DATA_BLOCK "DB00800_St_ConstAiRawData"   // DB800
TITLE = Static DB [SYSTEM CONSTANTS] — Analog Input Card Types, Ranges and Coefficients
{ S7_Optimized_Access := 'TRUE' }
AUTHOR : M_Gledhill
FAMILY : SysConstants
NAME : St_ConstAiRawData
VERSION : 1.0
// PRACTICAL SERIES AUTOMATION LIBRARY (PAL)   —   COPYRIGHT 2020 – M. GLEDHILL (MIT LICENCE)
//                   ———— ◆ ————
// FULL ONLINE DOCUMENTATION IS AVAILABLE AT: https://practicalseries.com/2001-pal/index.html
// stored: AutoNumber false, DBAccessibleFromOPCUA true, IsOnlyStoredInLoadMemory false, IsRetainMemResEnabled false, IsWriteProtectedInAS true, MemoryReserve 100
   VAR
      _DB_Header { ExternalAccessible := 'False'; ExternalVisible := 'False'; ExternalWritable := 'False'} : Array[0..79] of Bool;   // Static DB [SYSTEM CONSTANTS] — Analog Input Card Types, Ranges and Coefficients
      __________0000_0 { ExternalAccessible := 'False'; ExternalVisible := 'False'; ExternalWritable := 'False'} : Bool := false;
      __________0000_1 { ExternalAccessible := 'False'; ExternalVisible := 'False'; ExternalWritable := 'False'} : Bool := false;
      revInfo { ExternalWritable := 'False'} : "UT01000_St_SysRevision";
      __________0010_0 { ExternalAccessible := 'False'; ExternalVisible := 'False'; ExternalWritable := 'False'} : Bool := false;
      __________0010_1 { ExternalAccessible := 'False'; ExternalVisible := 'False'; ExternalWritable := 'False'} : Bool := false;
      AI_0000 { ExternalWritable := 'False'} : "UT00800_St_ConstAiRawData";
      __________0020_0 { ExternalAccessible := 'False'; ExternalVisible := 'False'; ExternalWritable := 'False'} : Bool := false;
      __________0020_1 { ExternalAccessible := 'False'; ExternalVisible := 'False'; ExternalWritable := 'False'} : Bool := false;   // ▀▀▀▀ ANALOG INPUT SIGNAL — VOLTAGE
      AI_1000 { ExternalWritable := 'False'} : "UT00800_St_ConstAiRawData";   // AI Voltage (-25 mV to +25 mV)
      AI_1001 { ExternalWritable := 'False'} : "UT00800_St_ConstAiRawData";   // AI Voltage (-50 mV to +50 mV)
      AI_1002 { ExternalWritable := 'False'} : "UT00800_St_ConstAiRawData";   // AI Voltage (-80 mV to +80 mV)
      AI_1003 { ExternalWritable := 'False'} : "UT00800_St_ConstAiRawData";   // AI Voltage (-250 mV to +250 mV)
      AI_1004 { ExternalWritable := 'False'} : "UT00800_St_ConstAiRawData";   // AI Voltage (-500 mV to +500 mV)
      AI_1005 { ExternalWritable := 'False'} : "UT00800_St_ConstAiRawData";   // AI Voltage (-1 V to +1 V)
      AI_1007 { ExternalWritable := 'False'} : "UT00800_St_ConstAiRawData";   // AI Voltage (-2.5 V to +2.5 V)
      AI_1008 { ExternalWritable := 'False'} : "UT00800_St_ConstAiRawData";   // AI Voltage (-5 V to +5 V)
      AI_1009 { ExternalWritable := 'False'} : "UT00800_St_ConstAiRawData";   // AI Voltage (-10 V to +10 V)
      AI_100A { ExternalWritable := 'False'} : "UT00800_St_ConstAiRawData";   // AI Voltage (1 V to 5 V)
      __________0030_0 { ExternalAccessible := 'False'; ExternalVisible := 'False'; ExternalWritable := 'False'} : Bool := false;
      __________0030_1 { ExternalAccessible := 'False'; ExternalVisible := 'False'; ExternalWritable := 'False'} : Bool := false;   // ▀▀▀▀ ANALOG INPUT SIGNAL — CURRENT (4 WIRE)
      AI_2002 { ExternalWritable := 'False'} : "UT00800_St_ConstAiRawData";   // AI Current - 4-wire (0 mA to 20 mA)
      AI_2003 { ExternalWritable := 'False'} : "UT00800_St_ConstAiRawData";   // AI Current - 4-wire (4 mA to 20 mA)
      AI_2004 { ExternalWritable := 'False'} : "UT00800_St_ConstAiRawData";   // AI Current - 4-wire (-20 mA to +20 mA)
      __________0040_0 { ExternalAccessible := 'False'; ExternalVisible := 'False'; ExternalWritable := 'False'} : Bool := false;
      __________0040_1 { ExternalAccessible := 'False'; ExternalVisible := 'False'; ExternalWritable := 'False'} : Bool := false;   // ▀▀▀▀ ANALOG INPUT SIGNAL — CURRENT (2 WIRE)
      AI_3003 { ExternalWritable := 'False'} : "UT00800_St_ConstAiRawData";   // AI Current - 2-wire (4 mA to 20 mA)
      __________0050_0 { ExternalAccessible := 'False'; ExternalVisible := 'False'; ExternalWritable := 'False'} : Bool := false;
      __________0050_1 { ExternalAccessible := 'False'; ExternalVisible := 'False'; ExternalWritable := 'False'} : Bool := false;   // ▀▀▀▀ ANALOG INPUT SIGNAL — RESISTANCE (4 WIRE)
      AI_4001 { ExternalWritable := 'False'} : "UT00800_St_ConstAiRawData";   // AI Resistance - 4-wire (150 Ohm)
      AI_4002 { ExternalWritable := 'False'} : "UT00800_St_ConstAiRawData";   // AI Resistance - 4-wire (300 Ohm)
      AI_4003 { ExternalWritable := 'False'} : "UT00800_St_ConstAiRawData";   // AI Resistance - 4-wire (600 Ohm)
      AI_4005 { ExternalWritable := 'False'} : "UT00800_St_ConstAiRawData";   // AI Resistance - 4-wire (6000 Ohm)
      __________0060_0 { ExternalAccessible := 'False'; ExternalVisible := 'False'; ExternalWritable := 'False'} : Bool := false;
      __________0060_1 { ExternalAccessible := 'False'; ExternalVisible := 'False'; ExternalWritable := 'False'} : Bool := false;   // ▀▀▀▀ ANALOG INPUT SIGNAL — RESISTANCE (3 WIRE)
      AI_5001 { ExternalWritable := 'False'} : "UT00800_St_ConstAiRawData";   // AI Resistance - 3-wire (150 Ohm)
      AI_5002 { ExternalWritable := 'False'} : "UT00800_St_ConstAiRawData";   // AI Resistance - 3-wire (300 Ohm)
      AI_5003 { ExternalWritable := 'False'} : "UT00800_St_ConstAiRawData";   // AI Resistance - 3-wire (600 Ohm)
      AI_5005 { ExternalWritable := 'False'} : "UT00800_St_ConstAiRawData";   // AI Resistance - 3-wire (6000 Ohm)
      __________0070_0 { ExternalAccessible := 'False'; ExternalVisible := 'False'; ExternalWritable := 'False'} : Bool := false;
      __________0070_1 { ExternalAccessible := 'False'; ExternalVisible := 'False'; ExternalWritable := 'False'} : Bool := false;   // ▀▀▀▀ ANALOG INPUT SIGNAL — RESISTANCE (2 WIRE)
      AI_6001 { ExternalWritable := 'False'} : "UT00800_St_ConstAiRawData";   // AI Resistance - 2-wire (150 Ohm)
      AI_6002 { ExternalWritable := 'False'} : "UT00800_St_ConstAiRawData";   // AI Resistance - 2-wire (300 Ohm)
      AI_6003 { ExternalWritable := 'False'} : "UT00800_St_ConstAiRawData";   // AI Resistance - 2-wire (600 Ohm)
      AI_6005 { ExternalWritable := 'False'} : "UT00800_St_ConstAiRawData";   // AI Resistance - 2-wire (6000 Ohm)
      AI_600F { ExternalWritable := 'False'} : "UT00800_St_ConstAiRawData";   // AI Resistance - 2-wire (PTC)
      __________0080_0 { ExternalAccessible := 'False'; ExternalVisible := 'False'; ExternalWritable := 'False'} : Bool := false;
      __________0080_1 { ExternalAccessible := 'False'; ExternalVisible := 'False'; ExternalWritable := 'False'} : Bool := false;   // ▀▀▀▀ ANALOG INPUT SIGNAL — THERMAL RESISTANCE (4 WIRE) Cu x0
      AI_7B0E { ExternalWritable := 'False'} : "UT00800_St_ConstAiRawData";   // AI Thermal Resistance - 4-wire (Cu10 climate - 426)
      AI_7C0E { ExternalWritable := 'False'} : "UT00800_St_ConstAiRawData";   // AI Thermal Resistance - 4-wire (Cu10 climate - 427)
      AI_7D0E { ExternalWritable := 'False'} : "UT00800_St_ConstAiRawData";   // AI Thermal Resistance - 4-wire (Cu10 climate - 428)
      AI_7B0F { ExternalWritable := 'False'} : "UT00800_St_ConstAiRawData";   // AI Thermal Resistance - 4-wire (Cu10 standard - 426)
      AI_7C0F { ExternalWritable := 'False'} : "UT00800_St_ConstAiRawData";   // AI Thermal Resistance - 4-wire (Cu10 standard - 427)
      AI_7D0F { ExternalWritable := 'False'} : "UT00800_St_ConstAiRawData";   // AI Thermal Resistance - 4-wire (Cu10 standard - 428)
      AI_7B19 { ExternalWritable := 'False'} : "UT00800_St_ConstAiRawData";   // AI Thermal Resistance - 4-wire (Cu50 climate - 426)
      AI_7C19 { ExternalWritable := 'False'} : "UT00800_St_ConstAiRawData";   // AI Thermal Resistance - 4-wire (Cu50 climate - 427)
      AI_7D19 { ExternalWritable := 'False'} : "UT00800_St_ConstAiRawData";   // AI Thermal Resistance - 4-wire (Cu50 climate - 428)
      AI_7B18 { ExternalWritable := 'False'} : "UT00800_St_ConstAiRawData";   // AI Thermal Resistance - 4-wire (Cu50 standard - 426)
      AI_7C18 { ExternalWritable := 'False'} : "UT00800_St_ConstAiRawData";   // AI Thermal Resistance - 4-wire (Cu50 standard - 427)
      AI_7D18 { ExternalWritable := 'False'} : "UT00800_St_ConstAiRawData";   // AI Thermal Resistance - 4-wire (Cu50 standard - 428)
      AI_7B1B { ExternalWritable := 'False'} : "UT00800_St_ConstAiRawData";   // AI Thermal Resistance - 4-wire (Cu100 climate - 426)
      AI_7C1B { ExternalWritable := 'False'} : "UT00800_St_ConstAiRawData";   // AI Thermal Resistance - 4-wire (Cu100 climate - 427)
      AI_7D1B { ExternalWritable := 'False'} : "UT00800_St_ConstAiRawData";   // AI Thermal Resistance - 4-wire (Cu100 climate - 428)
      AI_7B1A { ExternalWritable := 'False'} : "UT00800_St_ConstAiRawData";   // AI Thermal Resistance - 4-wire (Cu100 standard - 426)
      AI_7C1A { ExternalWritable := 'False'} : "UT00800_St_ConstAiRawData";   // AI Thermal Resistance - 4-wire (Cu100 standard - 427)
      AI_7D1A { ExternalWritable := 'False'} : "UT00800_St_ConstAiRawData";   // AI Thermal Resistance - 4-wire (Cu100 standard - 428)
      __________0090_0 { ExternalAccessible := 'False'; ExternalVisible := 'False'; ExternalWritable := 'False'} : Bool := false;
      __________0090_1 { ExternalAccessible := 'False'; ExternalVisible := 'False'; ExternalWritable := 'False'} : Bool := false;   // ▀▀▀▀ ANALOG INPUT SIGNAL — THERMAL RESISTANCE (4 WIRE) LG-Ni x0
      AI_7A1D { ExternalWritable := 'False'} : "UT00800_St_ConstAiRawData";   // AI Thermal Resistance - 4-wire (LG-Ni1000 climate - 500)
      AI_7A1C { ExternalWritable := 'False'} : "UT00800_St_ConstAiRawData";   // AI Thermal Resistance - 4-wire (LG-Ni1000 standard - 500)
      __________0100_0 { ExternalAccessible := 'False'; ExternalVisible := 'False'; ExternalWritable := 'False'} : Bool := false;
      __________0100_1 { ExternalAccessible := 'False'; ExternalVisible := 'False'; ExternalWritable := 'False'} : Bool := false;   // ▀▀▀▀ ANALOG INPUT SIGNAL — THERMAL RESISTANCE (4 WIRE) Ni x0
      AI_771F { ExternalWritable := 'False'} : "UT00800_St_ConstAiRawData";   // AI Thermal Resistance - 4-wire (Ni10 climate - 617)
      AI_781F { ExternalWritable := 'False'} : "UT00800_St_ConstAiRawData";   // AI Thermal Resistance - 4-wire (Ni10 climate - 618)
      AI_791F { ExternalWritable := 'False'} : "UT00800_St_ConstAiRawData";   // AI Thermal Resistance - 4-wire (Ni10 climate - 672)
      AI_771E { ExternalWritable := 'False'} : "UT00800_St_ConstAiRawData";   // AI Thermal Resistance - 4-wire (Ni10 standard - 617)
      AI_781E { ExternalWritable := 'False'} : "UT00800_St_ConstAiRawData";   // AI Thermal Resistance - 4-wire (Ni10 standard - 618)
      AI_791E { ExternalWritable := 'False'} : "UT00800_St_ConstAiRawData";   // AI Thermal Resistance - 4-wire (Ni10 standard - 672)
      AI_770D { ExternalWritable := 'False'} : "UT00800_St_ConstAiRawData";   // AI Thermal Resistance - 4-wire (Ni120 climate - 617)
      AI_780D { ExternalWritable := 'False'} : "UT00800_St_ConstAiRawData";   // AI Thermal Resistance - 4-wire (Ni120 climate - 618)
      AI_790D { ExternalWritable := 'False'} : "UT00800_St_ConstAiRawData";   // AI Thermal Resistance - 4-wire (Ni120 climate - 672)
      AI_770C { ExternalWritable := 'False'} : "UT00800_St_ConstAiRawData";   // AI Thermal Resistance - 4-wire (Ni120 standard - 617)
      AI_780C { ExternalWritable := 'False'} : "UT00800_St_ConstAiRawData";   // AI Thermal Resistance - 4-wire (Ni120 standard - 618)
      AI_790C { ExternalWritable := 'False'} : "UT00800_St_ConstAiRawData";   // AI Thermal Resistance - 4-wire (Ni120 standard - 672)
      AI_7701 { ExternalWritable := 'False'} : "UT00800_St_ConstAiRawData";   // AI Thermal Resistance - 4-wire (Ni100 climate - 617)
      AI_7801 { ExternalWritable := 'False'} : "UT00800_St_ConstAiRawData";   // AI Thermal Resistance - 4-wire (Ni100 climate - 618)
      AI_7901 { ExternalWritable := 'False'} : "UT00800_St_ConstAiRawData";   // AI Thermal Resistance - 4-wire (Ni100 climate - 672)
      AI_7703 { ExternalWritable := 'False'} : "UT00800_St_ConstAiRawData";   // AI Thermal Resistance - 4-wire (Ni100 standard - 617)
      AI_7803 { ExternalWritable := 'False'} : "UT00800_St_ConstAiRawData";   // AI Thermal Resistance - 4-wire (Ni100 standard - 618)
      AI_7903 { ExternalWritable := 'False'} : "UT00800_St_ConstAiRawData";   // AI Thermal Resistance - 4-wire (Ni100 standard - 672)
      AI_7711 { ExternalWritable := 'False'} : "UT00800_St_ConstAiRawData";   // AI Thermal Resistance - 4-wire (Ni200 climate - 617)
      AI_7811 { ExternalWritable := 'False'} : "UT00800_St_ConstAiRawData";   // AI Thermal Resistance - 4-wire (Ni200 climate - 618)
      AI_7911 { ExternalWritable := 'False'} : "UT00800_St_ConstAiRawData";   // AI Thermal Resistance - 4-wire (Ni200 climate - 672)
      AI_7710 { ExternalWritable := 'False'} : "UT00800_St_ConstAiRawData";   // AI Thermal Resistance - 4-wire (Ni200 standard - 617)
      AI_7810 { ExternalWritable := 'False'} : "UT00800_St_ConstAiRawData";   // AI Thermal Resistance - 4-wire (Ni200 standard - 618)
      AI_7910 { ExternalWritable := 'False'} : "UT00800_St_ConstAiRawData";   // AI Thermal Resistance - 4-wire (Ni200 standard - 672)
      AI_7713 { ExternalWritable := 'False'} : "UT00800_St_ConstAiRawData";   // AI Thermal Resistance - 4-wire (Ni500 climate - 617)
      AI_7813 { ExternalWritable := 'False'} : "UT00800_St_ConstAiRawData";   // AI Thermal Resistance - 4-wire (Ni500 climate - 618)
      AI_7913 { ExternalWritable := 'False'} : "UT00800_St_ConstAiRawData";   // AI Thermal Resistance - 4-wire (Ni500 climate - 672)
      AI_7712 { ExternalWritable := 'False'} : "UT00800_St_ConstAiRawData";   // AI Thermal Resistance - 4-wire (Ni500 standard - 617)
      AI_7812 { ExternalWritable := 'False'} : "UT00800_St_ConstAiRawData";   // AI Thermal Resistance - 4-wire (Ni500 standard - 618)
      AI_7912 { ExternalWritable := 'False'} : "UT00800_St_ConstAiRawData";   // AI Thermal Resistance - 4-wire (Ni500 standard - 672)
      AI_770A { ExternalWritable := 'False'} : "UT00800_St_ConstAiRawData";   // AI Thermal Resistance - 4-wire (Ni1000 climate - 617)
      AI_780A { ExternalWritable := 'False'} : "UT00800_St_ConstAiRawData";   // AI Thermal Resistance - 4-wire (Ni1000 climate - 618)
      AI_790A { ExternalWritable := 'False'} : "UT00800_St_ConstAiRawData";   // AI Thermal Resistance - 4-wire (Ni1000 climate - 672)
      AI_7706 { ExternalWritable := 'False'} : "UT00800_St_ConstAiRawData";   // AI Thermal Resistance - 4-wire (Ni1000 standard - 617)
      AI_7806 { ExternalWritable := 'False'} : "UT00800_St_ConstAiRawData";   // AI Thermal Resistance - 4-wire (Ni1000 standard - 618)
      AI_7906 { ExternalWritable := 'False'} : "UT00800_St_ConstAiRawData";   // AI Thermal Resistance - 4-wire (Ni1000 standard - 672)
      __________0110_0 { ExternalAccessible := 'False'; ExternalVisible := 'False'; ExternalWritable := 'False'} : Bool := false;
      __________0110_1 { ExternalAccessible := 'False'; ExternalVisible := 'False'; ExternalWritable := 'False'} : Bool := false;   // ▀▀▀▀ ANALOG INPUT SIGNAL — THERMAL RESISTANCE (4 WIRE) Pt x0
      AI_7015 { ExternalWritable := 'False'} : "UT00800_St_ConstAiRawData";   // AI Thermal Resistance - 4-wire (Pt10 climate - 3851)
      AI_7215 { ExternalWritable := 'False'} : "UT00800_St_ConstAiRawData";   // AI Thermal Resistance - 4-wire (Pt10 climate - 3902)
      AI_7515 { ExternalWritable := 'False'} : "UT00800_St_ConstAiRawData";   // AI Thermal Resistance - 4-wire (Pt10 climate - 391)
      AI_7115 { ExternalWritable := 'False'} : "UT00800_St_ConstAiRawData";   // AI Thermal Resistance - 4-wire (Pt10 climate - 3916)
      AI_7315 { ExternalWritable := 'False'} : "UT00800_St_ConstAiRawData";   // AI Thermal Resistance - 4-wire (Pt10 climate - 392)
      AI_7014 { ExternalWritable := 'False'} : "UT00800_St_ConstAiRawData";   // AI Thermal Resistance - 4-wire (Pt10 standard - 3851)
      AI_7214 { ExternalWritable := 'False'} : "UT00800_St_ConstAiRawData";   // AI Thermal Resistance - 4-wire (Pt10 standard - 3902)
      AI_7514 { ExternalWritable := 'False'} : "UT00800_St_ConstAiRawData";   // AI Thermal Resistance - 4-wire (Pt10 standard - 391)
      AI_7114 { ExternalWritable := 'False'} : "UT00800_St_ConstAiRawData";   // AI Thermal Resistance - 4-wire (Pt10 standard - 3916)
      AI_7314 { ExternalWritable := 'False'} : "UT00800_St_ConstAiRawData";   // AI Thermal Resistance - 4-wire (Pt10 standard - 392)
      AI_7017 { ExternalWritable := 'False'} : "UT00800_St_ConstAiRawData";   // AI Thermal Resistance - 4-wire (Pt50 climate - 3851)
      AI_7217 { ExternalWritable := 'False'} : "UT00800_St_ConstAiRawData";   // AI Thermal Resistance - 4-wire (Pt50 climate - 3902)
      AI_7517 { ExternalWritable := 'False'} : "UT00800_St_ConstAiRawData";   // AI Thermal Resistance - 4-wire (Pt50 climate - 391)
      AI_7117 { ExternalWritable := 'False'} : "UT00800_St_ConstAiRawData";   // AI Thermal Resistance - 4-wire (Pt50 climate - 3916)
      AI_7317 { ExternalWritable := 'False'} : "UT00800_St_ConstAiRawData";   // AI Thermal Resistance - 4-wire (Pt50 climate - 392)
      AI_7016 { ExternalWritable := 'False'} : "UT00800_St_ConstAiRawData";   // AI Thermal Resistance - 4-wire (Pt50 standard - 3851)
      AI_7216 { ExternalWritable := 'False'} : "UT00800_St_ConstAiRawData";   // AI Thermal Resistance - 4-wire (Pt50 standard - 3902)
      AI_7516 { ExternalWritable := 'False'} : "UT00800_St_ConstAiRawData";   // AI Thermal Resistance - 4-wire (Pt50 standard - 391)
      AI_7116 { ExternalWritable := 'False'} : "UT00800_St_ConstAiRawData";   // AI Thermal Resistance - 4-wire (Pt50 standard - 3916)
      AI_7316 { ExternalWritable := 'False'} : "UT00800_St_ConstAiRawData";   // AI Thermal Resistance - 4-wire (Pt50 standard - 392)
      AI_7000 { ExternalWritable := 'False'} : "UT00800_St_ConstAiRawData";   // AI Thermal Resistance - 4-wire (Pt100 climate - 3851)
      AI_7200 { ExternalWritable := 'False'} : "UT00800_St_ConstAiRawData";   // AI Thermal Resistance - 4-wire (Pt100 climate - 3902)
      AI_7500 { ExternalWritable := 'False'} : "UT00800_St_ConstAiRawData";   // AI Thermal Resistance - 4-wire (Pt100 climate - 391)
      AI_7100 { ExternalWritable := 'False'} : "UT00800_St_ConstAiRawData";   // AI Thermal Resistance - 4-wire (Pt100 climate - 3916)
      AI_7300 { ExternalWritable := 'False'} : "UT00800_St_ConstAiRawData";   // AI Thermal Resistance - 4-wire (Pt100 climate - 392)
      AI_7002 { ExternalWritable := 'False'} : "UT00800_St_ConstAiRawData";   // AI Thermal Resistance - 4-wire (Pt100 standard - 3851)
      AI_7202 { ExternalWritable := 'False'} : "UT00800_St_ConstAiRawData";   // AI Thermal Resistance - 4-wire (Pt100 standard - 3902)
      AI_7502 { ExternalWritable := 'False'} : "UT00800_St_ConstAiRawData";   // AI Thermal Resistance - 4-wire (Pt100 standard - 391)
      AI_7102 { ExternalWritable := 'False'} : "UT00800_St_ConstAiRawData";   // AI Thermal Resistance - 4-wire (Pt100 standard - 3916)
      AI_7302 { ExternalWritable := 'False'} : "UT00800_St_ConstAiRawData";   // AI Thermal Resistance - 4-wire (Pt100 standard - 392)
      AI_7007 { ExternalWritable := 'False'} : "UT00800_St_ConstAiRawData";   // AI Thermal Resistance - 4-wire (Pt200 climate - 3851)
      AI_7207 { ExternalWritable := 'False'} : "UT00800_St_ConstAiRawData";   // AI Thermal Resistance - 4-wire (Pt200 climate - 3902)
      AI_7507 { ExternalWritable := 'False'} : "UT00800_St_ConstAiRawData";   // AI Thermal Resistance - 4-wire (Pt200 climate - 391)
      AI_7107 { ExternalWritable := 'False'} : "UT00800_St_ConstAiRawData";   // AI Thermal Resistance - 4-wire (Pt200 climate - 3916)
      AI_7307 { ExternalWritable := 'False'} : "UT00800_St_ConstAiRawData";   // AI Thermal Resistance - 4-wire (Pt200 climate - 392)
      AI_700B { ExternalWritable := 'False'} : "UT00800_St_ConstAiRawData";   // AI Thermal Resistance - 4-wire (Pt200 standard - 3851)
      AI_720B { ExternalWritable := 'False'} : "UT00800_St_ConstAiRawData";   // AI Thermal Resistance - 4-wire (Pt200 standard - 3902)
      AI_750B { ExternalWritable := 'False'} : "UT00800_St_ConstAiRawData";   // AI Thermal Resistance - 4-wire (Pt200 standard - 391)
      AI_710B { ExternalWritable := 'False'} : "UT00800_St_ConstAiRawData";   // AI Thermal Resistance - 4-wire (Pt200 standard - 3916)
      AI_730B { ExternalWritable := 'False'} : "UT00800_St_ConstAiRawData";   // AI Thermal Resistance - 4-wire (Pt200 standard - 392)
      AI_7008 { ExternalWritable := 'False'} : "UT00800_St_ConstAiRawData";   // AI Thermal Resistance - 4-wire (Pt500 climate - 3851)
      AI_7208 { ExternalWritable := 'False'} : "UT00800_St_ConstAiRawData";   // AI Thermal Resistance - 4-wire (Pt500 climate - 3902)
      AI_7508 { ExternalWritable := 'False'} : "UT00800_St_ConstAiRawData";   // AI Thermal Resistance - 4-wire (Pt500 climate - 391)
      AI_7108 { ExternalWritable := 'False'} : "UT00800_St_ConstAiRawData";   // AI Thermal Resistance - 4-wire (Pt500 climate - 3916)
      AI_7308 { ExternalWritable := 'False'} : "UT00800_St_ConstAiRawData";   // AI Thermal Resistance - 4-wire (Pt500 climate - 392)
      AI_7004 { ExternalWritable := 'False'} : "UT00800_St_ConstAiRawData";   // AI Thermal Resistance - 4-wire (Pt500 standard - 3851)
      AI_7204 { ExternalWritable := 'False'} : "UT00800_St_ConstAiRawData";   // AI Thermal Resistance - 4-wire (Pt500 standard - 3902)
      AI_7504 { ExternalWritable := 'False'} : "UT00800_St_ConstAiRawData";   // AI Thermal Resistance - 4-wire (Pt500 standard - 391)
      AI_7104 { ExternalWritable := 'False'} : "UT00800_St_ConstAiRawData";   // AI Thermal Resistance - 4-wire (Pt500 standard - 3916)
      AI_7304 { ExternalWritable := 'False'} : "UT00800_St_ConstAiRawData";   // AI Thermal Resistance - 4-wire (Pt500 standard - 392)
      AI_7009 { ExternalWritable := 'False'} : "UT00800_St_ConstAiRawData";   // AI Thermal Resistance - 4-wire (Pt1000 climate - 3851)
      AI_7209 { ExternalWritable := 'False'} : "UT00800_St_ConstAiRawData";   // AI Thermal Resistance - 4-wire (Pt1000 climate - 3902)
      AI_7509 { ExternalWritable := 'False'} : "UT00800_St_ConstAiRawData";   // AI Thermal Resistance - 4-wire (Pt1000 climate - 391)
      AI_7109 { ExternalWritable := 'False'} : "UT00800_St_ConstAiRawData";   // AI Thermal Resistance - 4-wire (Pt1000 climate - 3916)
      AI_7309 { ExternalWritable := 'False'} : "UT00800_St_ConstAiRawData";   // AI Thermal Resistance - 4-wire (Pt1000 climate - 392)
      AI_7005 { ExternalWritable := 'False'} : "UT00800_St_ConstAiRawData";   // AI Thermal Resistance - 4-wire (Pt1000 standard - 3851)
      AI_7205 { ExternalWritable := 'False'} : "UT00800_St_ConstAiRawData";   // AI Thermal Resistance - 4-wire (Pt1000 standard - 3902)
      AI_7505 { ExternalWritable := 'False'} : "UT00800_St_ConstAiRawData";   // AI Thermal Resistance - 4-wire (Pt1000 standard - 391)
      AI_7105 { ExternalWritable := 'False'} : "UT00800_St_ConstAiRawData";   // AI Thermal Resistance - 4-wire (Pt1000 standard - 3916)
      AI_7305 { ExternalWritable := 'False'} : "UT00800_St_ConstAiRawData";   // AI Thermal Resistance - 4-wire (Pt1000 standard - 392)
      __________0120_0 { ExternalAccessible := 'False'; ExternalVisible := 'False'; ExternalWritable := 'False'} : Bool := false;
      __________0120_1 { ExternalAccessible := 'False'; ExternalVisible := 'False'; ExternalWritable := 'False'} : Bool := false;   // ▀▀▀▀ ANALOG INPUT SIGNAL — THERMAL RESISTANCE (3 WIRE) Cu x0
      AI_8B0E { ExternalWritable := 'False'} : "UT00800_St_ConstAiRawData";   // AI Thermal Resistance - 3-wire (Cu10 climate - 426)
      AI_8C0E { ExternalWritable := 'False'} : "UT00800_St_ConstAiRawData";   // AI Thermal Resistance - 3-wire (Cu10 climate - 427)
      AI_8D0E { ExternalWritable := 'False'} : "UT00800_St_ConstAiRawData";   // AI Thermal Resistance - 3-wire (Cu10 climate - 428)
      AI_8B0F { ExternalWritable := 'False'} : "UT00800_St_ConstAiRawData";   // AI Thermal Resistance - 3-wire (Cu10 standard - 426)
      AI_8C0F { ExternalWritable := 'False'} : "UT00800_St_ConstAiRawData";   // AI Thermal Resistance - 3-wire (Cu10 standard - 427)
      AI_8D0F { ExternalWritable := 'False'} : "UT00800_St_ConstAiRawData";   // AI Thermal Resistance - 3-wire (Cu10 standard - 428)
      AI_8B19 { ExternalWritable := 'False'} : "UT00800_St_ConstAiRawData";   // AI Thermal Resistance - 3-wire (Cu50 climate - 426)
      AI_8C19 { ExternalWritable := 'False'} : "UT00800_St_ConstAiRawData";   // AI Thermal Resistance - 3-wire (Cu50 climate - 427)
      AI_8D19 { ExternalWritable := 'False'} : "UT00800_St_ConstAiRawData";   // AI Thermal Resistance - 3-wire (Cu50 climate - 428)
      AI_8B18 { ExternalWritable := 'False'} : "UT00800_St_ConstAiRawData";   // AI Thermal Resistance - 3-wire (Cu50 standard - 426)
      AI_8C18 { ExternalWritable := 'False'} : "UT00800_St_ConstAiRawData";   // AI Thermal Resistance - 3-wire (Cu50 standard - 427)
      AI_8D18 { ExternalWritable := 'False'} : "UT00800_St_ConstAiRawData";   // AI Thermal Resistance - 3-wire (Cu50 standard - 428)
      AI_8B1B { ExternalWritable := 'False'} : "UT00800_St_ConstAiRawData";   // AI Thermal Resistance - 3-wire (Cu100 climate - 426)
      AI_8C1B { ExternalWritable := 'False'} : "UT00800_St_ConstAiRawData";   // AI Thermal Resistance - 3-wire (Cu100 climate - 427)
      AI_8D1B { ExternalWritable := 'False'} : "UT00800_St_ConstAiRawData";   // AI Thermal Resistance - 3-wire (Cu100 climate - 428)
      AI_8B1A { ExternalWritable := 'False'} : "UT00800_St_ConstAiRawData";   // AI Thermal Resistance - 3-wire (Cu100 standard - 426)
      AI_8C1A { ExternalWritable := 'False'} : "UT00800_St_ConstAiRawData";   // AI Thermal Resistance - 3-wire (Cu100 standard - 427)
      AI_8D1A { ExternalWritable := 'False'} : "UT00800_St_ConstAiRawData";   // AI Thermal Resistance - 3-wire (Cu100 standard - 428)
      __________0130_0 { ExternalAccessible := 'False'; ExternalVisible := 'False'; ExternalWritable := 'False'} : Bool := false;
      __________0130_1 { ExternalAccessible := 'False'; ExternalVisible := 'False'; ExternalWritable := 'False'} : Bool := false;   // ▀▀▀▀ ANALOG INPUT SIGNAL — THERMAL RESISTANCE (3 WIRE) LG-Ni x0
      AI_8A1D { ExternalWritable := 'False'} : "UT00800_St_ConstAiRawData";   // AI Thermal Resistance - 3-wire (LG-Ni1000 climate - 500)
      AI_8A1C { ExternalWritable := 'False'} : "UT00800_St_ConstAiRawData";   // AI Thermal Resistance - 3-wire (LG-Ni1000 standard - 500)
      __________0140_0 { ExternalAccessible := 'False'; ExternalVisible := 'False'; ExternalWritable := 'False'} : Bool := false;
      __________0140_1 { ExternalAccessible := 'False'; ExternalVisible := 'False'; ExternalWritable := 'False'} : Bool := false;   // ▀▀▀▀ ANALOG INPUT SIGNAL — THERMAL RESISTANCE (3 WIRE) Ni x0
      AI_871F { ExternalWritable := 'False'} : "UT00800_St_ConstAiRawData";   // AI Thermal Resistance - 3-wire (Ni10 climate - 617)
      AI_881F { ExternalWritable := 'False'} : "UT00800_St_ConstAiRawData";   // AI Thermal Resistance - 3-wire (Ni10 climate - 618)
      AI_891F { ExternalWritable := 'False'} : "UT00800_St_ConstAiRawData";   // AI Thermal Resistance - 3-wire (Ni10 climate - 672)
      AI_871E { ExternalWritable := 'False'} : "UT00800_St_ConstAiRawData";   // AI Thermal Resistance - 3-wire (Ni10 standard - 617)
      AI_881E { ExternalWritable := 'False'} : "UT00800_St_ConstAiRawData";   // AI Thermal Resistance - 3-wire (Ni10 standard - 618)
      AI_891E { ExternalWritable := 'False'} : "UT00800_St_ConstAiRawData";   // AI Thermal Resistance - 3-wire (Ni10 standard - 672)
      AI_870D { ExternalWritable := 'False'} : "UT00800_St_ConstAiRawData";   // AI Thermal Resistance - 3-wire (Ni120 climate - 617)
      AI_880D { ExternalWritable := 'False'} : "UT00800_St_ConstAiRawData";   // AI Thermal Resistance - 3-wire (Ni120 climate - 618)
      AI_890D { ExternalWritable := 'False'} : "UT00800_St_ConstAiRawData";   // AI Thermal Resistance - 3-wire (Ni120 climate - 672)
      AI_870C { ExternalWritable := 'False'} : "UT00800_St_ConstAiRawData";   // AI Thermal Resistance - 3-wire (Ni120 standard - 617)
      AI_880C { ExternalWritable := 'False'} : "UT00800_St_ConstAiRawData";   // AI Thermal Resistance - 3-wire (Ni120 standard - 618)
      AI_890C { ExternalWritable := 'False'} : "UT00800_St_ConstAiRawData";   // AI Thermal Resistance - 3-wire (Ni120 standard - 672)
      AI_8701 { ExternalWritable := 'False'} : "UT00800_St_ConstAiRawData";   // AI Thermal Resistance - 3-wire (Ni100 climate - 617)
      AI_8801 { ExternalWritable := 'False'} : "UT00800_St_ConstAiRawData";   // AI Thermal Resistance - 3-wire (Ni100 climate - 618)
      AI_8901 { ExternalWritable := 'False'} : "UT00800_St_ConstAiRawData";   // AI Thermal Resistance - 3-wire (Ni100 climate - 672)
      AI_8703 { ExternalWritable := 'False'} : "UT00800_St_ConstAiRawData";   // AI Thermal Resistance - 3-wire (Ni100 standard - 617)
      AI_8803 { ExternalWritable := 'False'} : "UT00800_St_ConstAiRawData";   // AI Thermal Resistance - 3-wire (Ni100 standard - 618)
      AI_8903 { ExternalWritable := 'False'} : "UT00800_St_ConstAiRawData";   // AI Thermal Resistance - 3-wire (Ni100 standard - 672)
      AI_8711 { ExternalWritable := 'False'} : "UT00800_St_ConstAiRawData";   // AI Thermal Resistance - 3-wire (Ni200 climate - 617)
      AI_8811 { ExternalWritable := 'False'} : "UT00800_St_ConstAiRawData";   // AI Thermal Resistance - 3-wire (Ni200 climate - 618)
      AI_8911 { ExternalWritable := 'False'} : "UT00800_St_ConstAiRawData";   // AI Thermal Resistance - 3-wire (Ni200 climate - 672)
      AI_8710 { ExternalWritable := 'False'} : "UT00800_St_ConstAiRawData";   // AI Thermal Resistance - 3-wire (Ni200 standard - 617)
      AI_8810 { ExternalWritable := 'False'} : "UT00800_St_ConstAiRawData";   // AI Thermal Resistance - 3-wire (Ni200 standard - 618)
      AI_8910 { ExternalWritable := 'False'} : "UT00800_St_ConstAiRawData";   // AI Thermal Resistance - 3-wire (Ni200 standard - 672)
      AI_8713 { ExternalWritable := 'False'} : "UT00800_St_ConstAiRawData";   // AI Thermal Resistance - 3-wire (Ni500 climate - 617)
      AI_8813 { ExternalWritable := 'False'} : "UT00800_St_ConstAiRawData";   // AI Thermal Resistance - 3-wire (Ni500 climate - 618)
      AI_8913 { ExternalWritable := 'False'} : "UT00800_St_ConstAiRawData";   // AI Thermal Resistance - 3-wire (Ni500 climate - 672)
      AI_8712 { ExternalWritable := 'False'} : "UT00800_St_ConstAiRawData";   // AI Thermal Resistance - 3-wire (Ni500 standard - 617)
      AI_8812 { ExternalWritable := 'False'} : "UT00800_St_ConstAiRawData";   // AI Thermal Resistance - 3-wire (Ni500 standard - 618)
      AI_8912 { ExternalWritable := 'False'} : "UT00800_St_ConstAiRawData";   // AI Thermal Resistance - 3-wire (Ni500 standard - 672)
      AI_870A { ExternalWritable := 'False'} : "UT00800_St_ConstAiRawData";   // AI Thermal Resistance - 3-wire (Ni1000 climate - 617)
      AI_880A { ExternalWritable := 'False'} : "UT00800_St_ConstAiRawData";   // AI Thermal Resistance - 3-wire (Ni1000 climate - 618)
      AI_890A { ExternalWritable := 'False'} : "UT00800_St_ConstAiRawData";   // AI Thermal Resistance - 3-wire (Ni1000 climate - 672)
      AI_8706 { ExternalWritable := 'False'} : "UT00800_St_ConstAiRawData";   // AI Thermal Resistance - 3-wire (Ni1000 standard - 617)
      AI_8806 { ExternalWritable := 'False'} : "UT00800_St_ConstAiRawData";   // AI Thermal Resistance - 3-wire (Ni1000 standard - 618)
      AI_8906 { ExternalWritable := 'False'} : "UT00800_St_ConstAiRawData";   // AI Thermal Resistance - 3-wire (Ni1000 standard - 672)
      __________0150_0 { ExternalAccessible := 'False'; ExternalVisible := 'False'; ExternalWritable := 'False'} : Bool := false;
      __________0150_1 { ExternalAccessible := 'False'; ExternalVisible := 'False'; ExternalWritable := 'False'} : Bool := false;   // ▀▀▀▀ ANALOG INPUT SIGNAL — THERMAL RESISTANCE (3 WIRE) Pt x0
      AI_8015 { ExternalWritable := 'False'} : "UT00800_St_ConstAiRawData";   // AI Thermal Resistance - 3-wire (Pt10 climate - 3851)
      AI_8215 { ExternalWritable := 'False'} : "UT00800_St_ConstAiRawData";   // AI Thermal Resistance - 3-wire (Pt10 climate - 3902)
      AI_8515 { ExternalWritable := 'False'} : "UT00800_St_ConstAiRawData";   // AI Thermal Resistance - 3-wire (Pt10 climate - 391)
      AI_8115 { ExternalWritable := 'False'} : "UT00800_St_ConstAiRawData";   // AI Thermal Resistance - 3-wire (Pt10 climate - 3916)
      AI_8315 { ExternalWritable := 'False'} : "UT00800_St_ConstAiRawData";   // AI Thermal Resistance - 3-wire (Pt10 climate - 392)
      AI_8014 { ExternalWritable := 'False'} : "UT00800_St_ConstAiRawData";   // AI Thermal Resistance - 3-wire (Pt10 standard - 3851)
      AI_8214 { ExternalWritable := 'False'} : "UT00800_St_ConstAiRawData";   // AI Thermal Resistance - 3-wire (Pt10 standard - 3902)
      AI_8514 { ExternalWritable := 'False'} : "UT00800_St_ConstAiRawData";   // AI Thermal Resistance - 3-wire (Pt10 standard - 391)
      AI_8114 { ExternalWritable := 'False'} : "UT00800_St_ConstAiRawData";   // AI Thermal Resistance - 3-wire (Pt10 standard - 3916)
      AI_8314 { ExternalWritable := 'False'} : "UT00800_St_ConstAiRawData";   // AI Thermal Resistance - 3-wire (Pt10 standard - 392)
      AI_8017 { ExternalWritable := 'False'} : "UT00800_St_ConstAiRawData";   // AI Thermal Resistance - 3-wire (Pt50 climate - 3851)
      AI_8217 { ExternalWritable := 'False'} : "UT00800_St_ConstAiRawData";   // AI Thermal Resistance - 3-wire (Pt50 climate - 3902)
      AI_8517 { ExternalWritable := 'False'} : "UT00800_St_ConstAiRawData";   // AI Thermal Resistance - 3-wire (Pt50 climate - 391)
      AI_8117 { ExternalWritable := 'False'} : "UT00800_St_ConstAiRawData";   // AI Thermal Resistance - 3-wire (Pt50 climate - 3916)
      AI_8317 { ExternalWritable := 'False'} : "UT00800_St_ConstAiRawData";   // AI Thermal Resistance - 3-wire (Pt50 climate - 392)
      AI_8016 { ExternalWritable := 'False'} : "UT00800_St_ConstAiRawData";   // AI Thermal Resistance - 3-wire (Pt50 standard - 3851)
      AI_8216 { ExternalWritable := 'False'} : "UT00800_St_ConstAiRawData";   // AI Thermal Resistance - 3-wire (Pt50 standard - 3902)
      AI_8516 { ExternalWritable := 'False'} : "UT00800_St_ConstAiRawData";   // AI Thermal Resistance - 3-wire (Pt50 standard - 391)
      AI_8116 { ExternalWritable := 'False'} : "UT00800_St_ConstAiRawData";   // AI Thermal Resistance - 3-wire (Pt50 standard - 3916)
      AI_8316 { ExternalWritable := 'False'} : "UT00800_St_ConstAiRawData";   // AI Thermal Resistance - 3-wire (Pt50 standard - 392)
      AI_8000 { ExternalWritable := 'False'} : "UT00800_St_ConstAiRawData";   // AI Thermal Resistance - 3-wire (Pt100 climate - 3851)
      AI_8200 { ExternalWritable := 'False'} : "UT00800_St_ConstAiRawData";   // AI Thermal Resistance - 3-wire (Pt100 climate - 3902)
      AI_8500 { ExternalWritable := 'False'} : "UT00800_St_ConstAiRawData";   // AI Thermal Resistance - 3-wire (Pt100 climate - 391)
      AI_8100 { ExternalWritable := 'False'} : "UT00800_St_ConstAiRawData";   // AI Thermal Resistance - 3-wire (Pt100 climate - 3916)
      AI_8300 { ExternalWritable := 'False'; S7_SetPoint := 'True'} : "UT00800_St_ConstAiRawData";   // AI Thermal Resistance - 3-wire (Pt100 climate - 392)
      AI_8002 { ExternalWritable := 'False'} : "UT00800_St_ConstAiRawData";   // AI Thermal Resistance - 3-wire (Pt100 standard - 3851)
   END_VAR
   VAR RETAIN
      AI_8202 { ExternalWritable := 'False'} : "UT00800_St_ConstAiRawData";   // AI Thermal Resistance - 3-wire (Pt100 standard - 3902)
   END_VAR
   VAR
      AI_8502 { ExternalWritable := 'False'} : "UT00800_St_ConstAiRawData";   // AI Thermal Resistance - 3-wire (Pt100 standard - 391)
      AI_8102 { ExternalWritable := 'False'} : "UT00800_St_ConstAiRawData";   // AI Thermal Resistance - 3-wire (Pt100 standard - 3916)
      AI_8302 { ExternalWritable := 'False'} : "UT00800_St_ConstAiRawData";   // AI Thermal Resistance - 3-wire (Pt100 standard - 392)
      AI_8007 { ExternalWritable := 'False'} : "UT00800_St_ConstAiRawData";   // AI Thermal Resistance - 3-wire (Pt200 climate - 3851)
      AI_8207 { ExternalWritable := 'False'} : "UT00800_St_ConstAiRawData";   // AI Thermal Resistance - 3-wire (Pt200 climate - 3902)
      AI_8507 { ExternalWritable := 'False'} : "UT00800_St_ConstAiRawData";   // AI Thermal Resistance - 3-wire (Pt200 climate - 391)
      AI_8107 { ExternalWritable := 'False'} : "UT00800_St_ConstAiRawData";   // AI Thermal Resistance - 3-wire (Pt200 climate - 3916)
      AI_8307 { ExternalWritable := 'False'} : "UT00800_St_ConstAiRawData";   // AI Thermal Resistance - 3-wire (Pt200 climate - 392)
      AI_800B { ExternalWritable := 'False'} : "UT00800_St_ConstAiRawData";   // AI Thermal Resistance - 3-wire (Pt200 standard - 3851)
      AI_820B { ExternalWritable := 'False'} : "UT00800_St_ConstAiRawData";   // AI Thermal Resistance - 3-wire (Pt200 standard - 3902)
      AI_850B { ExternalWritable := 'False'} : "UT00800_St_ConstAiRawData";   // AI Thermal Resistance - 3-wire (Pt200 standard - 391)
      AI_810B { ExternalWritable := 'False'} : "UT00800_St_ConstAiRawData";   // AI Thermal Resistance - 3-wire (Pt200 standard - 3916)
      AI_830B { ExternalWritable := 'False'} : "UT00800_St_ConstAiRawData";   // AI Thermal Resistance - 3-wire (Pt200 standard - 392)
      AI_8008 { ExternalWritable := 'False'} : "UT00800_St_ConstAiRawData";   // AI Thermal Resistance - 3-wire (Pt500 climate - 3851)
      AI_8208 { ExternalWritable := 'False'} : "UT00800_St_ConstAiRawData";   // AI Thermal Resistance - 3-wire (Pt500 climate - 3902)
      AI_8508 { ExternalWritable := 'False'} : "UT00800_St_ConstAiRawData";   // AI Thermal Resistance - 3-wire (Pt500 climate - 391)
      AI_8108 { ExternalWritable := 'False'} : "UT00800_St_ConstAiRawData";   // AI Thermal Resistance - 3-wire (Pt500 climate - 3916)
      AI_8308 { ExternalWritable := 'False'} : "UT00800_St_ConstAiRawData";   // AI Thermal Resistance - 3-wire (Pt500 climate - 392)
      AI_8004 { ExternalWritable := 'False'} : "UT00800_St_ConstAiRawData";   // AI Thermal Resistance - 3-wire (Pt500 standard - 3851)
      AI_8204 { ExternalWritable := 'False'} : "UT00800_St_ConstAiRawData";   // AI Thermal Resistance - 3-wire (Pt500 standard - 3902)
      AI_8504 { ExternalWritable := 'False'} : "UT00800_St_ConstAiRawData";   // AI Thermal Resistance - 3-wire (Pt500 standard - 391)
      AI_8104 { ExternalWritable := 'False'} : "UT00800_St_ConstAiRawData";   // AI Thermal Resistance - 3-wire (Pt500 standard - 3916)
      AI_8304 { ExternalWritable := 'False'} : "UT00800_St_ConstAiRawData";   // AI Thermal Resistance - 3-wire (Pt500 standard - 392)
      AI_8009 { ExternalWritable := 'False'} : "UT00800_St_ConstAiRawData";   // AI Thermal Resistance - 3-wire (Pt1000 climate - 3851)
      AI_8209 { ExternalWritable := 'False'} : "UT00800_St_ConstAiRawData";   // AI Thermal Resistance - 3-wire (Pt1000 climate - 3902)
      AI_8509 { ExternalWritable := 'False'} : "UT00800_St_ConstAiRawData";   // AI Thermal Resistance - 3-wire (Pt1000 climate - 391)
      AI_8109 { ExternalWritable := 'False'} : "UT00800_St_ConstAiRawData";   // AI Thermal Resistance - 3-wire (Pt1000 climate - 3916)
      AI_8309 { ExternalWritable := 'False'} : "UT00800_St_ConstAiRawData";   // AI Thermal Resistance - 3-wire (Pt1000 climate - 392)
      AI_8005 { ExternalWritable := 'False'} : "UT00800_St_ConstAiRawData";   // AI Thermal Resistance - 3-wire (Pt1000 standard - 3851)
      AI_8205 { ExternalWritable := 'False'} : "UT00800_St_ConstAiRawData";   // AI Thermal Resistance - 3-wire (Pt1000 standard - 3902)
      AI_8505 { ExternalWritable := 'False'} : "UT00800_St_ConstAiRawData";   // AI Thermal Resistance - 3-wire (Pt1000 standard - 391)
      AI_8105 { ExternalWritable := 'False'} : "UT00800_St_ConstAiRawData";   // AI Thermal Resistance - 3-wire (Pt1000 standard - 3916)
      AI_8305 { ExternalWritable := 'False'} : "UT00800_St_ConstAiRawData";   // AI Thermal Resistance - 3-wire (Pt1000 standard - 392)
      __________0160_0 { ExternalAccessible := 'False'; ExternalVisible := 'False'; ExternalWritable := 'False'} : Bool := false;
      __________0160_1 { ExternalAccessible := 'False'; ExternalVisible := 'False'; ExternalWritable := 'False'} : Bool := false;   // ▀▀▀▀ ANALOG INPUT SIGNAL — THERMOCOUPLE
      AI_A000 { ExternalWritable := 'False'} : "UT00800_St_ConstAiRawData";   // AI Thermocouple (Type B)
      AI_A00A { ExternalWritable := 'False'} : "UT00800_St_ConstAiRawData";   // AI Thermocouple (Type C)
      AI_A002 { ExternalWritable := 'False'} : "UT00800_St_ConstAiRawData";   // AI Thermocouple (Type E)
      AI_A005 { ExternalWritable := 'False'} : "UT00800_St_ConstAiRawData";   // AI Thermocouple (Type J)
      AI_A008 { ExternalWritable := 'False'} : "UT00800_St_ConstAiRawData";   // AI Thermocouple (Type K)
      AI_A001 { ExternalWritable := 'False'} : "UT00800_St_ConstAiRawData";   // AI Thermocouple (Type N)
      AI_A003 { ExternalWritable := 'False'} : "UT00800_St_ConstAiRawData";   // AI Thermocouple (Type R)
      AI_A004 { ExternalWritable := 'False'} : "UT00800_St_ConstAiRawData";   // AI Thermocouple (Type S)
      AI_A007 { ExternalWritable := 'False'} : "UT00800_St_ConstAiRawData";   // AI Thermocouple (Type T)
      AI_A00B { ExternalWritable := 'False'} : "UT00800_St_ConstAiRawData";   // AI Thermocouple (Type TXK/XCL)
   END_VAR
BEGIN
   // _DB_Header[0] : ▄▄▄▄▄▄▄▄▄▄▄▄▄▄▄▄▄▄▄▄▄▄▄▄▄▄▄▄▄▄▄▄ ＣＯＮＳＴＡＮＴＳ ▄▄
   // _DB_Header[2] : TITLE: SYSTEM CONSTANTS — ANALOG INPUT CARD TYPE, RANGE AND COEFFICIENTS
   // _DB_Header[4] : ▀▀▀▀▀▀▀▀▀▀▀▀▀▀▀▀▀▀▀▀▀▀▀▀▀▀▀▀▀▀▀▀▀▀▀▀▀▀▀▀▀▀▀▀
   // _DB_Header[5] : TYPE: STATIC
   // _DB_Header[6] : ▄▄▄▄▄▄▄▄▄▄▄▄▄▄▄▄▄▄▄▄▄▄▄▄▄▄▄▄▄▄▄▄▄▄▄▄▄▄▄▄▄▄▄▄
   // _DB_Header[8] : DB00800_St_ConstAiRawData is a static data block that holds a full set of range, parameter and
   // _DB_Header[9] : descriptive data for all types of analog input card channels.
   // _DB_Header[11] : Each dataset is stored in a structure of user data type: UT00800_St_ConstAiRawData.
   // _DB_Header[12] : This structure is configured to hold all the data required by the card itself, any module accessing
   // _DB_Header[13] : an analog input and any supervisory system that is to display the type and configuration of the
   // _DB_Header[14] : input channel.
   // _DB_Header[16] : All the channel data is stored as constants and is used by all modules that have an interface
   // _DB_Header[17] : to an analog input card.
   // _DB_Header[19] : The purpose of the user data type and associated data block is to provide a consistent and
   // _DB_Header[20] : tested set of range, parameter and descriptive data that can be used directly by modules that
   // _DB_Header[21] : interface with analog input cards.
   // _DB_Header[23] : The ranges correspond to the numerical values returned by the card for a given type of analog
   // _DB_Header[24] : card signal. For example, a 4-20 mA card returns a numerical value of 0 at 4 mA ranging up to a
   // _DB_Header[25] : value of 27648 at 20 mA. The data specified in the UT00800 variable would have a lower limit of
   // _DB_Header[26] : 0 and an upper limit of 27648.
   // _DB_Header[28] : In addition, each dataset contains the parametric data that defines the particular channel type
   // _DB_Header[29] : and can be used to set a particular analog input channel to a particular type and range during
   // _DB_Header[30] : runtime. Each dataset also contains a textual description of the channel type,:
   // _DB_Header[31] : e.g. Current – 4 wire (4 mA to 20 mA)
   // _DB_Header[32] : for display and information purposes.
   // _DB_Header[34] : Finally, data associated with thermal resistance channel types also contain the real number
   // _DB_Header[35] : value of the spe-cific temperature coefficient that is to be applied to the channel.
   // _DB_Header[37] : The PDF version of the SMDS for this module is available online here:
   // _DB_Header[38] : http://psop.uk/pal-smds-db00800-p
   // _DB_Header[40] : ━━━ ⬙⬙⬙⬙⬙⬙ ━━━
   // _DB_Header[42] : ▄▄▄▄▄▄▄▄▄▄▄▄▄▄▄▄▄▄▄▄▄▄▄▄▄▄▄▄▄▄▄▄▄▄▄▄▄▄▄▄▄▄▄▄
   // _DB_Header[43] : MODIFICATION HISTORY
   // _DB_Header[45] : This is a summary of the recent software modifications made to this block (most recent at top)
   // _DB_Header[47] : ―――――――――――――――――――――――――――――――――――――――――――
   // _DB_Header[48] : DATE REVISION MASTER BRANCH DEV
   // _DB_Header[49] : (nnn.amm) COMMIT TAG (Base ---> Merge) BRANCH Author
   // _DB_Header[50] : ———————————————————————————————————————————
   // _DB_Header[51] : 2024.05.07 001.000 D0017A-000.103 D0017 N/A D0017A M. Gledhill
   // _DB_Header[52] : DB00800 — RELEASED FOR USE
   // _DB_Header[54] : 2024.05.03 000.801 D0017A-000.102 D0017 N/A D0017A M. Gledhill
   // _DB_Header[55] : DB00800 Block populated
   // _DB_Header[56] : 2024.04.09 000.101 D0017A-000.101 D0017 N/A D0017A M. Gledhill
   // _DB_Header[57] : DB00800 Block created
   // _DB_Header[58] : ———————————————————————————————————————————
   // _DB_Header[59] : Where: nnn = Major revision
   // _DB_Header[60] : a = Type (1-7 Development, 8 Proving, 9 Qualification, 0 Release)
   // _DB_Header[61] : mm = Minor revision (must be 00 if a = 0)
   // _DB_Header[62] : Block properties version number should be set to nn.a (only one decimal place)
   // _DB_Header[64] : ██████████████ █ █ █ █ END █ █ █ █ ██████████████
   revInfo.REV_BLOCK := 'DB00800';
   revInfo.REV_NUMBER := '000.801';
   revInfo.REV_DATE := '2024-05-03';
   revInfo.REV_AUTHOR := 'M. Gledhill';
   AI_0000.AI_CODE := 16#0000;
   AI_0000.___________0020_0 := false;
   AI_0000.___________0010_2 := false;
   AI_0000.RAW_MIN := 0;
   AI_0000.RAW_MAX := 0;
   AI_0000.RAW_NAME := 'User defined signal type';
   AI_0000.___________0030_1 := false;
   AI_0000.___________0030_2 := false;
   AI_0000.PARAM_TYPE := 16#00;
   AI_0000.PARAM_RANGE := 16#00;
   AI_0000.PARAM_COEF := 16#00;
   AI_1000.AI_CODE := 16#1000;
   AI_1000.___________0020_0 := false;
   AI_1000.___________0010_2 := false;
   AI_1000.RAW_MIN := -27648;
   AI_1000.RAW_MAX := 27648;
   AI_1000.RAW_NAME := 'Voltage (-25 mV to +25 mV)';
   AI_1000.___________0030_1 := false;
   AI_1000.___________0030_2 := false;
   AI_1000.PARAM_TYPE := 16#01;
   AI_1000.PARAM_RANGE := 16#00;
   AI_1000.PARAM_COEF := 16#00;
   AI_1001.AI_CODE := 16#1001;
   AI_1001.___________0020_0 := false;
   AI_1001.___________0010_2 := false;
   AI_1001.RAW_MIN := -27648;
   AI_1001.RAW_MAX := 27648;
   AI_1001.RAW_NAME := 'Voltage (-50 mV to +50 mV)';
   AI_1001.___________0030_1 := false;
   AI_1001.___________0030_2 := false;
   AI_1001.PARAM_TYPE := 16#01;
   AI_1001.PARAM_RANGE := 16#01;
   AI_1001.PARAM_COEF := 16#00;
   AI_1002.AI_CODE := 16#1002;
   AI_1002.___________0020_0 := false;
   AI_1002.___________0010_2 := false;
   AI_1002.RAW_MIN := -27648;
   AI_1002.RAW_MAX := 27648;
   AI_1002.RAW_NAME := 'Voltage (-80 mV to +80 mV)';
   AI_1002.___________0030_1 := false;
   AI_1002.___________0030_2 := false;
   AI_1002.PARAM_TYPE := 16#01;
   AI_1002.PARAM_RANGE := 16#02;
   AI_1002.PARAM_COEF := 16#00;
   AI_1003.AI_CODE := 16#1003;
   AI_1003.___________0020_0 := false;
   AI_1003.___________0010_2 := false;
   AI_1003.RAW_MIN := -27648;
   AI_1003.RAW_MAX := 27648;
   AI_1003.RAW_NAME := 'Voltage (-250 mV to +250 mV)';
   AI_1003.___________0030_1 := false;
   AI_1003.___________0030_2 := false;
   AI_1003.PARAM_TYPE := 16#01;
   AI_1003.PARAM_RANGE := 16#03;
   AI_1003.PARAM_COEF := 16#00;
   AI_1004.AI_CODE := 16#1004;
   AI_1004.___________0020_0 := false;
   AI_1004.___________0010_2 := false;
   AI_1004.RAW_MIN := -27648;
   AI_1004.RAW_MAX := 27648;
   AI_1004.RAW_NAME := 'Voltage (-500 mV to +500 mV)';
   AI_1004.___________0030_1 := false;
   AI_1004.___________0030_2 := false;
   AI_1004.PARAM_TYPE := 16#01;
   AI_1004.PARAM_RANGE := 16#04;
   AI_1004.PARAM_COEF := 16#00;
   AI_1005.AI_CODE := 16#1005;
   AI_1005.___________0020_0 := false;
   AI_1005.___________0010_2 := false;
   AI_1005.RAW_MIN := -27648;
   AI_1005.RAW_MAX := 27648;
   AI_1005.RAW_NAME := 'Voltage (-1 V to +1 V)';
   AI_1005.___________0030_1 := false;
   AI_1005.___________0030_2 := false;
   AI_1005.PARAM_TYPE := 16#01;
   AI_1005.PARAM_RANGE := 16#05;
   AI_1005.PARAM_COEF := 16#00;
   AI_1007.AI_CODE := 16#1007;
   AI_1007.___________0020_0 := false;
   AI_1007.___________0010_2 := false;
   AI_1007.RAW_MIN := -27648;
   AI_1007.RAW_MAX := 27648;
   AI_1007.RAW_NAME := 'Voltage (-2.5 V to +2.5 V)';
   AI_1007.___________0030_1 := false;
   AI_1007.___________0030_2 := false;
   AI_1007.PARAM_TYPE := 16#01;
   AI_1007.PARAM_RANGE := 16#07;
   AI_1007.PARAM_COEF := 16#00;
   AI_1008.AI_CODE := 16#1008;
   AI_1008.___________0020_0 := false;
   AI_1008.___________0010_2 := false;
   AI_1008.RAW_MIN := -27648;
   AI_1008.RAW_MAX := 27648;
   AI_1008.RAW_NAME := 'Voltage (-5 V to +5 V)';
   AI_1008.___________0030_1 := false;
   AI_1008.___________0030_2 := false;
   AI_1008.PARAM_TYPE := 16#01;
   AI_1008.PARAM_RANGE := 16#08;
   AI_1008.PARAM_COEF := 16#00;
   AI_1009.AI_CODE := 16#1009;
   AI_1009.___________0020_0 := false;
   AI_1009.___________0010_2 := false;
   AI_1009.RAW_MIN := -27648;
   AI_1009.RAW_MAX := 27648;
   AI_1009.RAW_NAME := 'Voltage (-10 V to +10 V)';
   AI_1009.___________0030_1 := false;
   AI_1009.___________0030_2 := false;
   AI_1009.PARAM_TYPE := 16#01;
   AI_1009.PARAM_RANGE := 16#09;
   AI_1009.PARAM_COEF := 16#00;
   AI_100A.AI_CODE := 16#100A;
   AI_100A.___________0020_0 := false;
   AI_100A.___________0010_2 := false;
   AI_100A.RAW_MIN := 0;
   AI_100A.RAW_MAX := 27648;
   AI_100A.RAW_NAME := 'Voltage (1 V to 5 V)';
   AI_100A.___________0030_1 := false;
   AI_100A.___________0030_2 := false;
   AI_100A.PARAM_TYPE := 16#01;
   AI_100A.PARAM_RANGE := 16#0A;
   AI_100A.PARAM_COEF := 16#00;
   AI_2002.AI_CODE := 16#2002;
   AI_2002.___________0020_0 := false;
   AI_2002.___________0010_2 := false;
   AI_2002.RAW_MIN := 0;
   AI_2002.RAW_MAX := 27648;
   AI_2002.RAW_NAME := 'Current - 4-wire (0 mA to 20 mA)';
   AI_2002.___________0030_1 := false;
   AI_2002.___________0030_2 := false;
   AI_2002.PARAM_TYPE := 16#02;
   AI_2002.PARAM_RANGE := 16#02;
   AI_2002.PARAM_COEF := 16#00;
   AI_2003.AI_CODE := 16#2003;
   AI_2003.___________0020_0 := false;
   AI_2003.___________0010_2 := false;
   AI_2003.RAW_MIN := 0;
   AI_2003.RAW_MAX := 27648;
   AI_2003.RAW_NAME := 'Current - 4-wire (4 mA to 20 mA)';
   AI_2003.___________0030_1 := false;
   AI_2003.___________0030_2 := false;
   AI_2003.PARAM_TYPE := 16#02;
   AI_2003.PARAM_RANGE := 16#03;
   AI_2003.PARAM_COEF := 16#00;
   AI_2004.AI_CODE := 16#2004;
   AI_2004.___________0020_0 := false;
   AI_2004.___________0010_2 := false;
   AI_2004.RAW_MIN := -27648;
   AI_2004.RAW_MAX := 27648;
   AI_2004.RAW_NAME := 'Current - 4-wire (-20 mA to +20 mA)';
   AI_2004.___________0030_1 := false;
   AI_2004.___________0030_2 := false;
   AI_2004.PARAM_TYPE := 16#02;
   AI_2004.PARAM_RANGE := 16#04;
   AI_2004.PARAM_COEF := 16#00;
   AI_3003.AI_CODE := 16#3003;
   AI_3003.___________0020_0 := false;
   AI_3003.___________0010_2 := false;
   AI_3003.RAW_MIN := 0;
   AI_3003.RAW_MAX := 27648;
   AI_3003.RAW_NAME := 'Current - 2-wire (4 mA to 20 mA)';
   AI_3003.___________0030_1 := false;
   AI_3003.___________0030_2 := false;
   AI_3003.PARAM_TYPE := 16#03;
   AI_3003.PARAM_RANGE := 16#03;
   AI_3003.PARAM_COEF := 16#00;
   AI_4001.AI_CODE := 16#4001;
   AI_4001.___________0020_0 := false;
   AI_4001.___________0010_2 := false;
   AI_4001.RAW_MIN := 0;
   AI_4001.RAW_MAX := 27648;
   AI_4001.RAW_NAME := 'Resistance - 4-wire (150 Ohm)';
   AI_4001.___________0030_1 := false;
   AI_4001.___________0030_2 := false;
   AI_4001.PARAM_TYPE := 16#04;
   AI_4001.PARAM_RANGE := 16#01;
   AI_4001.PARAM_COEF := 16#00;
   AI_4002.AI_CODE := 16#4002;
   AI_4002.___________0020_0 := false;
   AI_4002.___________0010_2 := false;
   AI_4002.RAW_MIN := 0;
   AI_4002.RAW_MAX := 27648;
   AI_4002.RAW_NAME := 'Resistance - 4-wire (300 Ohm)';
   AI_4002.___________0030_1 := false;
   AI_4002.___________0030_2 := false;
   AI_4002.PARAM_TYPE := 16#04;
   AI_4002.PARAM_RANGE := 16#02;
   AI_4002.PARAM_COEF := 16#00;
   AI_4003.AI_CODE := 16#4003;
   AI_4003.___________0020_0 := false;
   AI_4003.___________0010_2 := false;
   AI_4003.RAW_MIN := 0;
   AI_4003.RAW_MAX := 27648;
   AI_4003.RAW_NAME := 'Resistance - 4-wire (600 Ohm)';
   AI_4003.___________0030_1 := false;
   AI_4003.___________0030_2 := false;
   AI_4003.PARAM_TYPE := 16#04;
   AI_4003.PARAM_RANGE := 16#03;
   AI_4003.PARAM_COEF := 16#00;
   AI_4005.AI_CODE := 16#4005;
   AI_4005.___________0020_0 := false;
   AI_4005.___________0010_2 := false;
   AI_4005.RAW_MIN := 0;
   AI_4005.RAW_MAX := 27648;
   AI_4005.RAW_NAME := 'Resistance - 4-wire (6000 Ohm)';
   AI_4005.___________0030_1 := false;
   AI_4005.___________0030_2 := false;
   AI_4005.PARAM_TYPE := 16#04;
   AI_4005.PARAM_RANGE := 16#05;
   AI_4005.PARAM_COEF := 16#00;
   AI_5001.AI_CODE := 16#5001;
   AI_5001.___________0020_0 := false;
   AI_5001.___________0010_2 := false;
   AI_5001.RAW_MIN := 0;
   AI_5001.RAW_MAX := 27648;
   AI_5001.RAW_NAME := 'Resistance - 3-wire (150 Ohm)';
   AI_5001.___________0030_1 := false;
   AI_5001.___________0030_2 := false;
   AI_5001.PARAM_TYPE := 16#05;
   AI_5001.PARAM_RANGE := 16#01;
   AI_5001.PARAM_COEF := 16#00;
   AI_5002.AI_CODE := 16#5002;
   AI_5002.___________0020_0 := false;
   AI_5002.___________0010_2 := false;
   AI_5002.RAW_MIN := 0;
   AI_5002.RAW_MAX := 27648;
   AI_5002.RAW_NAME := 'Resistance - 3-wire (300 Ohm)';
   AI_5002.___________0030_1 := false;
   AI_5002.___________0030_2 := false;
   AI_5002.PARAM_TYPE := 16#05;
   AI_5002.PARAM_RANGE := 16#02;
   AI_5002.PARAM_COEF := 16#00;
   AI_5003.AI_CODE := 16#5003;
   AI_5003.___________0020_0 := false;
   AI_5003.___________0010_2 := false;
   AI_5003.RAW_MIN := 0;
   AI_5003.RAW_MAX := 27648;
   AI_5003.RAW_NAME := 'Resistance - 3-wire (600 Ohm)';
   AI_5003.___________0030_1 := false;
   AI_5003.___________0030_2 := false;
   AI_5003.PARAM_TYPE := 16#05;
   AI_5003.PARAM_RANGE := 16#03;
   AI_5003.PARAM_COEF := 16#00;
   AI_5005.AI_CODE := 16#5005;
   AI_5005.___________0020_0 := false;
   AI_5005.___________0010_2 := false;
   AI_5005.RAW_MIN := 0;
   AI_5005.RAW_MAX := 27648;
   AI_5005.RAW_NAME := 'Resistance - 3-wire (6000 Ohm)';
   AI_5005.___________0030_1 := false;
   AI_5005.___________0030_2 := false;
   AI_5005.PARAM_TYPE := 16#05;
   AI_5005.PARAM_RANGE := 16#05;
   AI_5005.PARAM_COEF := 16#00;
   AI_6001.AI_CODE := 16#6001;
   AI_6001.___________0020_0 := false;
   AI_6001.___________0010_2 := false;
   AI_6001.RAW_MIN := 0;
   AI_6001.RAW_MAX := 27648;
   AI_6001.RAW_NAME := 'Resistance - 2-wire (150 Ohm)';
   AI_6001.___________0030_1 := false;
   AI_6001.___________0030_2 := false;
   AI_6001.PARAM_TYPE := 16#06;
   AI_6001.PARAM_RANGE := 16#01;
   AI_6001.PARAM_COEF := 16#00;
   AI_6002.AI_CODE := 16#6002;
   AI_6002.___________0020_0 := false;
   AI_6002.___________0010_2 := false;
   AI_6002.RAW_MIN := 0;
   AI_6002.RAW_MAX := 27648;
   AI_6002.RAW_NAME := 'Resistance - 2-wire (300 Ohm)';
   AI_6002.___________0030_1 := false;
   AI_6002.___________0030_2 := false;
   AI_6002.PARAM_TYPE := 16#06;
   AI_6002.PARAM_RANGE := 16#02;
   AI_6002.PARAM_COEF := 16#00;
   AI_6003.AI_CODE := 16#6003;
   AI_6003.___________0020_0 := false;
   AI_6003.___________0010_2 := false;
   AI_6003.RAW_MIN := 0;
   AI_6003.RAW_MAX := 27648;
   AI_6003.RAW_NAME := 'Resistance - 2-wire (600 Ohm)';
   AI_6003.___________0030_1 := false;
   AI_6003.___________0030_2 := false;
   AI_6003.PARAM_TYPE := 16#06;
   AI_6003.PARAM_RANGE := 16#03;
   AI_6003.PARAM_COEF := 16#00;
   AI_6005.AI_CODE := 16#6005;
   AI_6005.___________0020_0 := false;
   AI_6005.___________0010_2 := false;
   AI_6005.RAW_MIN := 0;
   AI_6005.RAW_MAX := 27648;
   AI_6005.RAW_NAME := 'Resistance - 2-wire (6000 Ohm)';
   AI_6005.___________0030_1 := false;
   AI_6005.___________0030_2 := false;
   AI_6005.PARAM_TYPE := 16#06;
   AI_6005.PARAM_RANGE := 16#05;
   AI_6005.PARAM_COEF := 16#00;
   AI_600F.AI_CODE := 16#600F;
   AI_600F.___________0020_0 := false;
   AI_600F.___________0010_2 := false;
   AI_600F.RAW_MIN := 0;
   AI_600F.RAW_MAX := 27648;
   AI_600F.RAW_NAME := 'Resistance - 2-wire (PTC)';
   AI_600F.___________0030_1 := false;
   AI_600F.___________0030_2 := false;
   AI_600F.PARAM_TYPE := 16#06;
   AI_600F.PARAM_RANGE := 16#0F;
   AI_600F.PARAM_COEF := 16#00;
   AI_7B0E.AI_CODE := 16#7B0E;
   AI_7B0E.___________0020_0 := false;
   AI_7B0E.___________0010_2 := false;
   AI_7B0E.RAW_MIN := -5000;
   AI_7B0E.RAW_MAX := 15000;
   AI_7B0E.RAW_NAME := 'Thermal Resistance - 4-wire (Cu10 climate - 426)';
   AI_7B0E.___________0030_1 := false;
   AI_7B0E.___________0030_2 := false;
   AI_7B0E.PARAM_TYPE := 16#07;
   AI_7B0E.PARAM_RANGE := 16#0E;
   AI_7B0E.PARAM_COEF := 16#0B;
   AI_7B0E.VALUE_COEF := 0.00426;
   AI_7C0E.AI_CODE := 16#7C0E;
   AI_7C0E.___________0020_0 := false;
   AI_7C0E.___________0010_2 := false;
   AI_7C0E.RAW_MIN := -5000;
   AI_7C0E.RAW_MAX := 15000;
   AI_7C0E.RAW_NAME := 'Thermal Resistance - 4-wire (Cu10 climate - 427)';
   AI_7C0E.___________0030_1 := false;
   AI_7C0E.___________0030_2 := false;
   AI_7C0E.PARAM_TYPE := 16#07;
   AI_7C0E.PARAM_RANGE := 16#0E;
   AI_7C0E.PARAM_COEF := 16#0C;
   AI_7C0E.VALUE_COEF := 0.00427;
   AI_7D0E.AI_CODE := 16#7D0E;
   AI_7D0E.___________0020_0 := false;
   AI_7D0E.___________0010_2 := false;
   AI_7D0E.RAW_MIN := -5000;
   AI_7D0E.RAW_MAX := 15000;
   AI_7D0E.RAW_NAME := 'Thermal Resistance - 4-wire (Cu10 climate - 428)';
   AI_7D0E.___________0030_1 := false;
   AI_7D0E.___________0030_2 := false;
   AI_7D0E.PARAM_TYPE := 16#07;
   AI_7D0E.PARAM_RANGE := 16#0E;
   AI_7D0E.PARAM_COEF := 16#0D;
   AI_7D0E.VALUE_COEF := 0.00428;
   AI_7B0F.AI_CODE := 16#7B0F;
   AI_7B0F.___________0020_0 := false;
   AI_7B0F.___________0010_2 := false;
   AI_7B0F.RAW_MIN := -500;
   AI_7B0F.RAW_MAX := 2000;
   AI_7B0F.RAW_NAME := 'Thermal Resistance - 4-wire (Cu10 standard - 426)';
   AI_7B0F.___________0030_1 := false;
   AI_7B0F.___________0030_2 := false;
   AI_7B0F.PARAM_TYPE := 16#07;
   AI_7B0F.PARAM_RANGE := 16#0F;
   AI_7B0F.PARAM_COEF := 16#0B;
   AI_7B0F.VALUE_COEF := 0.00426;
   AI_7C0F.AI_CODE := 16#7C0F;
   AI_7C0F.___________0020_0 := false;
   AI_7C0F.___________0010_2 := false;
   AI_7C0F.RAW_MIN := -2000;
   AI_7C0F.RAW_MAX := 2600;
   AI_7C0F.RAW_NAME := 'Thermal Resistance - 4-wire (Cu10 standard - 427)';
   AI_7C0F.___________0030_1 := false;
   AI_7C0F.___________0030_2 := false;
   AI_7C0F.PARAM_TYPE := 16#07;
   AI_7C0F.PARAM_RANGE := 16#0F;
   AI_7C0F.PARAM_COEF := 16#0C;
   AI_7C0F.VALUE_COEF := 0.00427;
   AI_7D0F.AI_CODE := 16#7D0F;
   AI_7D0F.___________0020_0 := false;
   AI_7D0F.___________0010_2 := false;
   AI_7D0F.RAW_MIN := -1800;
   AI_7D0F.RAW_MAX := 2000;
   AI_7D0F.RAW_NAME := 'Thermal Resistance - 4-wire (Cu10 standard - 428)';
   AI_7D0F.___________0030_1 := false;
   AI_7D0F.___________0030_2 := false;
   AI_7D0F.PARAM_TYPE := 16#07;
   AI_7D0F.PARAM_RANGE := 16#0F;
   AI_7D0F.PARAM_COEF := 16#0D;
   AI_7D0F.VALUE_COEF := 0.00428;
   AI_7B19.AI_CODE := 16#7B19;
   AI_7B19.___________0020_0 := false;
   AI_7B19.___________0010_2 := false;
   AI_7B19.RAW_MIN := -5000;
   AI_7B19.RAW_MAX := 15000;
   AI_7B19.RAW_NAME := 'Thermal Resistance - 4-wire (Cu50 climate - 426)';
   AI_7B19.___________0030_1 := false;
   AI_7B19.___________0030_2 := false;
   AI_7B19.PARAM_TYPE := 16#07;
   AI_7B19.PARAM_RANGE := 16#19;
   AI_7B19.PARAM_COEF := 16#0B;
   AI_7B19.VALUE_COEF := 0.00426;
   AI_7C19.AI_CODE := 16#7C19;
   AI_7C19.___________0020_0 := false;
   AI_7C19.___________0010_2 := false;
   AI_7C19.RAW_MIN := -5000;
   AI_7C19.RAW_MAX := 15000;
   AI_7C19.RAW_NAME := 'Thermal Resistance - 4-wire (Cu50 climate - 427)';
   AI_7C19.___________0030_1 := false;
   AI_7C19.___________0030_2 := false;
   AI_7C19.PARAM_TYPE := 16#07;
   AI_7C19.PARAM_RANGE := 16#19;
   AI_7C19.PARAM_COEF := 16#0C;
   AI_7C19.VALUE_COEF := 0.00427;
   AI_7D19.AI_CODE := 16#7D19;
   AI_7D19.___________0020_0 := false;
   AI_7D19.___________0010_2 := false;
   AI_7D19.RAW_MIN := -5000;
   AI_7D19.RAW_MAX := 15000;
   AI_7D19.RAW_NAME := 'Thermal Resistance - 4-wire (Cu50 climate - 428)';
   AI_7D19.___________0030_1 := false;
   AI_7D19.___________0030_2 := false;
   AI_7D19.PARAM_TYPE := 16#07;
   AI_7D19.PARAM_RANGE := 16#19;
   AI_7D19.PARAM_COEF := 16#0D;
   AI_7D19.VALUE_COEF := 0.00428;
   AI_7B18.AI_CODE := 16#7B18;
   AI_7B18.___________0020_0 := false;
   AI_7B18.___________0010_2 := false;
   AI_7B18.RAW_MIN := -500;
   AI_7B18.RAW_MAX := 2000;
   AI_7B18.RAW_NAME := 'Thermal Resistance - 4-wire (Cu50 standard - 426)';
   AI_7B18.___________0030_1 := false;
   AI_7B18.___________0030_2 := false;
   AI_7B18.PARAM_TYPE := 16#07;
   AI_7B18.PARAM_RANGE := 16#18;
   AI_7B18.PARAM_COEF := 16#0B;
   AI_7B18.VALUE_COEF := 0.00426;
   AI_7C18.AI_CODE := 16#7C18;
   AI_7C18.___________0020_0 := false;
   AI_7C18.___________0010_2 := false;
   AI_7C18.RAW_MIN := -2000;
   AI_7C18.RAW_MAX := 2600;
   AI_7C18.RAW_NAME := 'Thermal Resistance - 4-wire (Cu50 standard - 427)';
   AI_7C18.___________0030_1 := false;
   AI_7C18.___________0030_2 := false;
   AI_7C18.PARAM_TYPE := 16#07;
   AI_7C18.PARAM_RANGE := 16#18;
   AI_7C18.PARAM_COEF := 16#0C;
   AI_7C18.VALUE_COEF := 0.00427;
   AI_7D18.AI_CODE := 16#7D18;
   AI_7D18.___________0020_0 := false;
   AI_7D18.___________0010_2 := false;
   AI_7D18.RAW_MIN := -1800;
   AI_7D18.RAW_MAX := 2000;
   AI_7D18.RAW_NAME := 'Thermal Resistance - 4-wire (Cu50 standard - 428)';
   AI_7D18.___________0030_1 := false;
   AI_7D18.___________0030_2 := false;
   AI_7D18.PARAM_TYPE := 16#07;
   AI_7D18.PARAM_RANGE := 16#18;
   AI_7D18.PARAM_COEF := 16#0D;
   AI_7D18.VALUE_COEF := 0.00428;
   AI_7B1B.AI_CODE := 16#7B1B;
   AI_7B1B.___________0020_0 := false;
   AI_7B1B.___________0010_2 := false;
   AI_7B1B.RAW_MIN := -5000;
   AI_7B1B.RAW_MAX := 15000;
   AI_7B1B.RAW_NAME := 'Thermal Resistance - 4-wire (Cu100 climate - 426)';
   AI_7B1B.___________0030_1 := false;
   AI_7B1B.___________0030_2 := false;
   AI_7B1B.PARAM_TYPE := 16#07;
   AI_7B1B.PARAM_RANGE := 16#1B;
   AI_7B1B.PARAM_COEF := 16#0B;
   AI_7B1B.VALUE_COEF := 0.00426;
   AI_7C1B.AI_CODE := 16#7C1B;
   AI_7C1B.___________0020_0 := false;
   AI_7C1B.___________0010_2 := false;
   AI_7C1B.RAW_MIN := -5000;
   AI_7C1B.RAW_MAX := 15000;
   AI_7C1B.RAW_NAME := 'Thermal Resistance - 4-wire (Cu100 climate - 427)';
   AI_7C1B.___________0030_1 := false;
   AI_7C1B.___________0030_2 := false;
   AI_7C1B.PARAM_TYPE := 16#07;
   AI_7C1B.PARAM_RANGE := 16#1B;
   AI_7C1B.PARAM_COEF := 16#0C;
   AI_7C1B.VALUE_COEF := 0.00427;
   AI_7D1B.AI_CODE := 16#7D1B;
   AI_7D1B.___________0020_0 := false;
   AI_7D1B.___________0010_2 := false;
   AI_7D1B.RAW_MIN := -5000;
   AI_7D1B.RAW_MAX := 15000;
   AI_7D1B.RAW_NAME := 'Thermal Resistance - 4-wire (Cu100 climate - 428)';
   AI_7D1B.___________0030_1 := false;
   AI_7D1B.___________0030_2 := false;
   AI_7D1B.PARAM_TYPE := 16#07;
   AI_7D1B.PARAM_RANGE := 16#1B;
   AI_7D1B.PARAM_COEF := 16#0D;
   AI_7D1B.VALUE_COEF := 0.00428;
   AI_7B1A.AI_CODE := 16#7B1A;
   AI_7B1A.___________0020_0 := false;
   AI_7B1A.___________0010_2 := false;
   AI_7B1A.RAW_MIN := -500;
   AI_7B1A.RAW_MAX := 2000;
   AI_7B1A.RAW_NAME := 'Thermal Resistance - 4-wire (Cu100 standard - 426)';
   AI_7B1A.___________0030_1 := false;
   AI_7B1A.___________0030_2 := false;
   AI_7B1A.PARAM_TYPE := 16#07;
   AI_7B1A.PARAM_RANGE := 16#1A;
   AI_7B1A.PARAM_COEF := 16#0B;
   AI_7B1A.VALUE_COEF := 0.00426;
   AI_7C1A.AI_CODE := 16#7C1A;
   AI_7C1A.___________0020_0 := false;
   AI_7C1A.___________0010_2 := false;
   AI_7C1A.RAW_MIN := -2000;
   AI_7C1A.RAW_MAX := 2600;
   AI_7C1A.RAW_NAME := 'Thermal Resistance - 4-wire (Cu100 standard - 427)';
   AI_7C1A.___________0030_1 := false;
   AI_7C1A.___________0030_2 := false;
   AI_7C1A.PARAM_TYPE := 16#07;
   AI_7C1A.PARAM_RANGE := 16#1A;
   AI_7C1A.PARAM_COEF := 16#0C;
   AI_7C1A.VALUE_COEF := 0.00427;
   AI_7D1A.AI_CODE := 16#7D1A;
   AI_7D1A.___________0020_0 := false;
   AI_7D1A.___________0010_2 := false;
   AI_7D1A.RAW_MIN := -1800;
   AI_7D1A.RAW_MAX := 2000;
   AI_7D1A.RAW_NAME := 'Thermal Resistance - 4-wire (Cu100 standard - 428)';
   AI_7D1A.___________0030_1 := false;
   AI_7D1A.___________0030_2 := false;
   AI_7D1A.PARAM_TYPE := 16#07;
   AI_7D1A.PARAM_RANGE := 16#1A;
   AI_7D1A.PARAM_COEF := 16#0D;
   AI_7D1A.VALUE_COEF := 0.00428;
   AI_7A1D.AI_CODE := 16#7A1D;
   AI_7A1D.___________0020_0 := false;
   AI_7A1D.___________0010_2 := false;
   AI_7A1D.RAW_MIN := -6000;
   AI_7A1D.RAW_MAX := 13000;
   AI_7A1D.RAW_NAME := 'Thermal Resistance - 4-wire (LG-Ni1000 climate - 500)';
   AI_7A1D.___________0030_1 := false;
   AI_7A1D.___________0030_2 := false;
   AI_7A1D.PARAM_TYPE := 16#07;
   AI_7A1D.PARAM_RANGE := 16#1D;
   AI_7A1D.PARAM_COEF := 16#0A;
   AI_7A1D.VALUE_COEF := 0.005;
   AI_7A1C.AI_CODE := 16#7A1C;
   AI_7A1C.___________0020_0 := false;
   AI_7A1C.___________0010_2 := false;
   AI_7A1C.RAW_MIN := -600;
   AI_7A1C.RAW_MAX := 2500;
   AI_7A1C.RAW_NAME := 'Thermal Resistance - 4-wire (LG-Ni1000 standard - 500)';
   AI_7A1C.___________0030_1 := false;
   AI_7A1C.___________0030_2 := false;
   AI_7A1C.PARAM_TYPE := 16#07;
   AI_7A1C.PARAM_RANGE := 16#1C;
   AI_7A1C.PARAM_COEF := 16#0A;
   AI_7A1C.VALUE_COEF := 0.005;
   AI_771F.AI_CODE := 16#771F;
   AI_771F.___________0020_0 := false;
   AI_771F.___________0010_2 := false;
   AI_771F.RAW_MIN := -6000;
   AI_771F.RAW_MAX := 13000;
   AI_771F.RAW_NAME := 'Thermal Resistance - 4-wire (Ni10 climate - 617)';
   AI_771F.___________0030_1 := false;
   AI_771F.___________0030_2 := false;
   AI_771F.PARAM_TYPE := 16#07;
   AI_771F.PARAM_RANGE := 16#1F;
   AI_771F.PARAM_COEF := 16#07;
   AI_771F.VALUE_COEF := 0.00617;
   AI_781F.AI_CODE := 16#781F;
   AI_781F.___________0020_0 := false;
   AI_781F.___________0010_2 := false;
   AI_781F.RAW_MIN := -6000;
   AI_781F.RAW_MAX := 13000;
   AI_781F.RAW_NAME := 'Thermal Resistance - 4-wire (Ni10 climate - 618)';
   AI_781F.___________0030_1 := false;
   AI_781F.___________0030_2 := false;
   AI_781F.PARAM_TYPE := 16#07;
   AI_781F.PARAM_RANGE := 16#1F;
   AI_781F.PARAM_COEF := 16#08;
   AI_781F.VALUE_COEF := 0.00618;
   AI_791F.AI_CODE := 16#791F;
   AI_791F.___________0020_0 := false;
   AI_791F.___________0010_2 := false;
   AI_791F.RAW_MIN := -6000;
   AI_791F.RAW_MAX := 13000;
   AI_791F.RAW_NAME := 'Thermal Resistance - 4-wire (Ni10 climate - 672)';
   AI_791F.___________0030_1 := false;
   AI_791F.___________0030_2 := false;
   AI_791F.PARAM_TYPE := 16#07;
   AI_791F.PARAM_RANGE := 16#1F;
   AI_791F.PARAM_COEF := 16#09;
   AI_791F.VALUE_COEF := 0.00672;
   AI_771E.AI_CODE := 16#771E;
   AI_771E.___________0020_0 := false;
   AI_771E.___________0010_2 := false;
   AI_771E.RAW_MIN := -600;
   AI_771E.RAW_MAX := 1800;
   AI_771E.RAW_NAME := 'Thermal Resistance - 4-wire (Ni10 standard - 617)';
   AI_771E.___________0030_1 := false;
   AI_771E.___________0030_2 := false;
   AI_771E.PARAM_TYPE := 16#07;
   AI_771E.PARAM_RANGE := 16#1E;
   AI_771E.PARAM_COEF := 16#07;
   AI_771E.VALUE_COEF := 0.00617;
   AI_781E.AI_CODE := 16#781E;
   AI_781E.___________0020_0 := false;
   AI_781E.___________0010_2 := false;
   AI_781E.RAW_MIN := -600;
   AI_781E.RAW_MAX := 2500;
   AI_781E.RAW_NAME := 'Thermal Resistance - 4-wire (Ni10 standard - 618)';
   AI_781E.___________0030_1 := false;
   AI_781E.___________0030_2 := false;
   AI_781E.PARAM_TYPE := 16#07;
   AI_781E.PARAM_RANGE := 16#1E;
   AI_781E.PARAM_COEF := 16#08;
   AI_781E.VALUE_COEF := 0.00618;
   AI_791E.AI_CODE := 16#791E;
   AI_791E.___________0020_0 := false;
   AI_791E.___________0010_2 := false;
   AI_791E.RAW_MIN := -600;
   AI_791E.RAW_MAX := 2500;
   AI_791E.RAW_NAME := 'Thermal Resistance - 4-wire (Ni10 standard - 672)';
   AI_791E.___________0030_1 := false;
   AI_791E.___________0030_2 := false;
   AI_791E.PARAM_TYPE := 16#07;
   AI_791E.PARAM_RANGE := 16#1E;
   AI_791E.PARAM_COEF := 16#09;
   AI_791E.VALUE_COEF := 0.00672;
   AI_770D.AI_CODE := 16#770D;
   AI_770D.___________0020_0 := false;
   AI_770D.___________0010_2 := false;
   AI_770D.RAW_MIN := -6000;
   AI_770D.RAW_MAX := 13000;
   AI_770D.RAW_NAME := 'Thermal Resistance - 4-wire (Ni120 climate - 617)';
   AI_770D.___________0030_1 := false;
   AI_770D.___________0030_2 := false;
   AI_770D.PARAM_TYPE := 16#07;
   AI_770D.PARAM_RANGE := 16#0D;
   AI_770D.PARAM_COEF := 16#07;
   AI_770D.VALUE_COEF := 0.00617;
   AI_780D.AI_CODE := 16#780D;
   AI_780D.___________0020_0 := false;
   AI_780D.___________0010_2 := false;
   AI_780D.RAW_MIN := -6000;
   AI_780D.RAW_MAX := 13000;
   AI_780D.RAW_NAME := 'Thermal Resistance - 4-wire (Ni120 climate - 618)';
   AI_780D.___________0030_1 := false;
   AI_780D.___________0030_2 := false;
   AI_780D.PARAM_TYPE := 16#07;
   AI_780D.PARAM_RANGE := 16#0D;
   AI_780D.PARAM_COEF := 16#08;
   AI_780D.VALUE_COEF := 0.00618;
   AI_790D.AI_CODE := 16#790D;
   AI_790D.___________0020_0 := false;
   AI_790D.___________0010_2 := false;
   AI_790D.RAW_MIN := -6000;
   AI_790D.RAW_MAX := 13000;
   AI_790D.RAW_NAME := 'Thermal Resistance - 4-wire (Ni120 climate - 672)';
   AI_790D.___________0030_1 := false;
   AI_790D.___________0030_2 := false;
   AI_790D.PARAM_TYPE := 16#07;
   AI_790D.PARAM_RANGE := 16#0D;
   AI_790D.PARAM_COEF := 16#09;
   AI_790D.VALUE_COEF := 0.00672;
   AI_770C.AI_CODE := 16#770C;
   AI_770C.___________0020_0 := false;
   AI_770C.___________0010_2 := false;
   AI_770C.RAW_MIN := -600;
   AI_770C.RAW_MAX := 1800;
   AI_770C.RAW_NAME := 'Thermal Resistance - 4-wire (Ni120 standard - 617)';
   AI_770C.___________0030_1 := false;
   AI_770C.___________0030_2 := false;
   AI_770C.PARAM_TYPE := 16#07;
   AI_770C.PARAM_RANGE := 16#0C;
   AI_770C.PARAM_COEF := 16#07;
   AI_770C.VALUE_COEF := 0.00617;
   AI_780C.AI_CODE := 16#780C;
   AI_780C.___________0020_0 := false;
   AI_780C.___________0010_2 := false;
   AI_780C.RAW_MIN := -600;
   AI_780C.RAW_MAX := 2500;
   AI_780C.RAW_NAME := 'Thermal Resistance - 4-wire (Ni120 standard - 618)';
   AI_780C.___________0030_1 := false;
   AI_780C.___________0030_2 := false;
   AI_780C.PARAM_TYPE := 16#07;
   AI_780C.PARAM_RANGE := 16#0C;
   AI_780C.PARAM_COEF := 16#08;
   AI_780C.VALUE_COEF := 0.00618;
   AI_790C.AI_CODE := 16#790C;
   AI_790C.___________0020_0 := false;
   AI_790C.___________0010_2 := false;
   AI_790C.RAW_MIN := -600;
   AI_790C.RAW_MAX := 2500;
   AI_790C.RAW_NAME := 'Thermal Resistance - 4-wire (Ni120 standard - 672)';
   AI_790C.___________0030_1 := false;
   AI_790C.___________0030_2 := false;
   AI_790C.PARAM_TYPE := 16#07;
   AI_790C.PARAM_RANGE := 16#0C;
   AI_790C.PARAM_COEF := 16#09;
   AI_790C.VALUE_COEF := 0.00672;
   AI_7701.AI_CODE := 16#7701;
   AI_7701.___________0020_0 := false;
   AI_7701.___________0010_2 := false;
   AI_7701.RAW_MIN := -6000;
   AI_7701.RAW_MAX := 13000;
   AI_7701.RAW_NAME := 'Thermal Resistance - 4-wire (Ni100 climate - 617)';
   AI_7701.___________0030_1 := false;
   AI_7701.___________0030_2 := false;
   AI_7701.PARAM_TYPE := 16#07;
   AI_7701.PARAM_RANGE := 16#01;
   AI_7701.PARAM_COEF := 16#07;
   AI_7701.VALUE_COEF := 0.00617;
   AI_7801.AI_CODE := 16#7801;
   AI_7801.___________0020_0 := false;
   AI_7801.___________0010_2 := false;
   AI_7801.RAW_MIN := -6000;
   AI_7801.RAW_MAX := 13000;
   AI_7801.RAW_NAME := 'Thermal Resistance - 4-wire (Ni100 climate - 618)';
   AI_7801.___________0030_1 := false;
   AI_7801.___________0030_2 := false;
   AI_7801.PARAM_TYPE := 16#07;
   AI_7801.PARAM_RANGE := 16#01;
   AI_7801.PARAM_COEF := 16#08;
   AI_7801.VALUE_COEF := 0.00618;
   AI_7901.AI_CODE := 16#7901;
   AI_7901.___________0020_0 := false;
   AI_7901.___________0010_2 := false;
   AI_7901.RAW_MIN := -6000;
   AI_7901.RAW_MAX := 13000;
   AI_7901.RAW_NAME := 'Thermal Resistance - 4-wire (Ni100 climate - 672)';
   AI_7901.___________0030_1 := false;
   AI_7901.___________0030_2 := false;
   AI_7901.PARAM_TYPE := 16#07;
   AI_7901.PARAM_RANGE := 16#01;
   AI_7901.PARAM_COEF := 16#09;
   AI_7901.VALUE_COEF := 0.00672;
   AI_7703.AI_CODE := 16#7703;
   AI_7703.___________0020_0 := false;
   AI_7703.___________0010_2 := false;
   AI_7703.RAW_MIN := -600;
   AI_7703.RAW_MAX := 1800;
   AI_7703.RAW_NAME := 'Thermal Resistance - 4-wire (Ni100 standard - 617)';
   AI_7703.___________0030_1 := false;
   AI_7703.___________0030_2 := false;
   AI_7703.PARAM_TYPE := 16#07;
   AI_7703.PARAM_RANGE := 16#03;
   AI_7703.PARAM_COEF := 16#07;
   AI_7703.VALUE_COEF := 0.00617;
   AI_7803.AI_CODE := 16#7803;
   AI_7803.___________0020_0 := false;
   AI_7803.___________0010_2 := false;
   AI_7803.RAW_MIN := -600;
   AI_7803.RAW_MAX := 2500;
   AI_7803.RAW_NAME := 'Thermal Resistance - 4-wire (Ni100 standard - 618)';
   AI_7803.___________0030_1 := false;
   AI_7803.___________0030_2 := false;
   AI_7803.PARAM_TYPE := 16#07;
   AI_7803.PARAM_RANGE := 16#03;
   AI_7803.PARAM_COEF := 16#08;
   AI_7803.VALUE_COEF := 0.00618;
   AI_7903.AI_CODE := 16#7903;
   AI_7903.___________0020_0 := false;
   AI_7903.___________0010_2 := false;
   AI_7903.RAW_MIN := -600;
   AI_7903.RAW_MAX := 2500;
   AI_7903.RAW_NAME := 'Thermal Resistance - 4-wire (Ni100 standard - 672)';
   AI_7903.___________0030_1 := false;
   AI_7903.___________0030_2 := false;
   AI_7903.PARAM_TYPE := 16#07;
   AI_7903.PARAM_RANGE := 16#03;
   AI_7903.PARAM_COEF := 16#09;
   AI_7903.VALUE_COEF := 0.00672;
   AI_7711.AI_CODE := 16#7711;
   AI_7711.___________0020_0 := false;
   AI_7711.___________0010_2 := false;
   AI_7711.RAW_MIN := -6000;
   AI_7711.RAW_MAX := 13000;
   AI_7711.RAW_NAME := 'Thermal Resistance - 4-wire (Ni200 climate - 617)';
   AI_7711.___________0030_1 := false;
   AI_7711.___________0030_2 := false;
   AI_7711.PARAM_TYPE := 16#07;
   AI_7711.PARAM_RANGE := 16#11;
   AI_7711.PARAM_COEF := 16#07;
   AI_7711.VALUE_COEF := 0.00617;
   AI_7811.AI_CODE := 16#7811;
   AI_7811.___________0020_0 := false;
   AI_7811.___________0010_2 := false;
   AI_7811.RAW_MIN := -6000;
   AI_7811.RAW_MAX := 13000;
   AI_7811.RAW_NAME := 'Thermal Resistance - 4-wire (Ni200 climate - 618)';
   AI_7811.___________0030_1 := false;
   AI_7811.___________0030_2 := false;
   AI_7811.PARAM_TYPE := 16#07;
   AI_7811.PARAM_RANGE := 16#11;
   AI_7811.PARAM_COEF := 16#08;
   AI_7811.VALUE_COEF := 0.00618;
   AI_7911.AI_CODE := 16#7911;
   AI_7911.___________0020_0 := false;
   AI_7911.___________0010_2 := false;
   AI_7911.RAW_MIN := -6000;
   AI_7911.RAW_MAX := 13000;
   AI_7911.RAW_NAME := 'Thermal Resistance - 4-wire (Ni200 climate - 672)';
   AI_7911.___________0030_1 := false;
   AI_7911.___________0030_2 := false;
   AI_7911.PARAM_TYPE := 16#07;
   AI_7911.PARAM_RANGE := 16#11;
   AI_7911.PARAM_COEF := 16#09;
   AI_7911.VALUE_COEF := 0.00672;
   AI_7710.AI_CODE := 16#7710;
   AI_7710.___________0020_0 := false;
   AI_7710.___________0010_2 := false;
   AI_7710.RAW_MIN := -600;
   AI_7710.RAW_MAX := 1800;
   AI_7710.RAW_NAME := 'Thermal Resistance - 4-wire (Ni200 standard - 617)';
   AI_7710.___________0030_1 := false;
   AI_7710.___________0030_2 := false;
   AI_7710.PARAM_TYPE := 16#07;
   AI_7710.PARAM_RANGE := 16#10;
   AI_7710.PARAM_COEF := 16#07;
   AI_7710.VALUE_COEF := 0.00617;
   AI_7810.AI_CODE := 16#7810;
   AI_7810.___________0020_0 := false;
   AI_7810.___________0010_2 := false;
   AI_7810.RAW_MIN := -600;
   AI_7810.RAW_MAX := 2500;
   AI_7810.RAW_NAME := 'Thermal Resistance - 4-wire (Ni200 standard - 618)';
   AI_7810.___________0030_1 := false;
   AI_7810.___________0030_2 := false;
   AI_7810.PARAM_TYPE := 16#07;
   AI_7810.PARAM_RANGE := 16#10;
   AI_7810.PARAM_COEF := 16#08;
   AI_7810.VALUE_COEF := 0.00618;
   AI_7910.AI_CODE := 16#7910;
   AI_7910.___________0020_0 := false;
   AI_7910.___________0010_2 := false;
   AI_7910.RAW_MIN := -600;
   AI_7910.RAW_MAX := 2500;
   AI_7910.RAW_NAME := 'Thermal Resistance - 4-wire (Ni200 standard - 672)';
   AI_7910.___________0030_1 := false;
   AI_7910.___________0030_2 := false;
   AI_7910.PARAM_TYPE := 16#07;
   AI_7910.PARAM_RANGE := 16#10;
   AI_7910.PARAM_COEF := 16#09;
   AI_7910.VALUE_COEF := 0.00672;
   AI_7713.AI_CODE := 16#7713;
   AI_7713.___________0020_0 := false;
   AI_7713.___________0010_2 := false;
   AI_7713.RAW_MIN := -6000;
   AI_7713.RAW_MAX := 13000;
   AI_7713.RAW_NAME := 'Thermal Resistance - 4-wire (Ni500 climate - 617)';
   AI_7713.___________0030_1 := false;
   AI_7713.___________0030_2 := false;
   AI_7713.PARAM_TYPE := 16#07;
   AI_7713.PARAM_RANGE := 16#13;
   AI_7713.PARAM_COEF := 16#07;
   AI_7713.VALUE_COEF := 0.00617;
   AI_7813.AI_CODE := 16#7813;
   AI_7813.___________0020_0 := false;
   AI_7813.___________0010_2 := false;
   AI_7813.RAW_MIN := -6000;
   AI_7813.RAW_MAX := 13000;
   AI_7813.RAW_NAME := 'Thermal Resistance - 4-wire (Ni500 climate - 618)';
   AI_7813.___________0030_1 := false;
   AI_7813.___________0030_2 := false;
   AI_7813.PARAM_TYPE := 16#07;
   AI_7813.PARAM_RANGE := 16#13;
   AI_7813.PARAM_COEF := 16#08;
   AI_7813.VALUE_COEF := 0.00618;
   AI_7913.AI_CODE := 16#7913;
   AI_7913.___________0020_0 := false;
   AI_7913.___________0010_2 := false;
   AI_7913.RAW_MIN := -6000;
   AI_7913.RAW_MAX := 13000;
   AI_7913.RAW_NAME := 'Thermal Resistance - 4-wire (Ni500 climate - 672)';
   AI_7913.___________0030_1 := false;
   AI_7913.___________0030_2 := false;
   AI_7913.PARAM_TYPE := 16#07;
   AI_7913.PARAM_RANGE := 16#13;
   AI_7913.PARAM_COEF := 16#09;
   AI_7913.VALUE_COEF := 0.00672;
   AI_7712.AI_CODE := 16#7712;
   AI_7712.___________0020_0 := false;
   AI_7712.___________0010_2 := false;
   AI_7712.RAW_MIN := -600;
   AI_7712.RAW_MAX := 1800;
   AI_7712.RAW_NAME := 'Thermal Resistance - 4-wire (Ni500 standard - 617)';
   AI_7712.___________0030_1 := false;
   AI_7712.___________0030_2 := false;
   AI_7712.PARAM_TYPE := 16#07;
   AI_7712.PARAM_RANGE := 16#12;
   AI_7712.PARAM_COEF := 16#07;
   AI_7712.VALUE_COEF := 0.00617;
   AI_7812.AI_CODE := 16#7812;
   AI_7812.___________0020_0 := false;
   AI_7812.___________0010_2 := false;
   AI_7812.RAW_MIN := -600;
   AI_7812.RAW_MAX := 2500;
   AI_7812.RAW_NAME := 'Thermal Resistance - 4-wire (Ni500 standard - 618)';
   AI_7812.___________0030_1 := false;
   AI_7812.___________0030_2 := false;
   AI_7812.PARAM_TYPE := 16#07;
   AI_7812.PARAM_RANGE := 16#12;
   AI_7812.PARAM_COEF := 16#08;
   AI_7812.VALUE_COEF := 0.00618;
   AI_7912.AI_CODE := 16#7912;
   AI_7912.___________0020_0 := false;
   AI_7912.___________0010_2 := false;
   AI_7912.RAW_MIN := -600;
   AI_7912.RAW_MAX := 2500;
   AI_7912.RAW_NAME := 'Thermal Resistance - 4-wire (Ni500 standard - 672)';
   AI_7912.___________0030_1 := false;
   AI_7912.___________0030_2 := false;
   AI_7912.PARAM_TYPE := 16#07;
   AI_7912.PARAM_RANGE := 16#12;
   AI_7912.PARAM_COEF := 16#09;
   AI_7912.VALUE_COEF := 0.00672;
   AI_770A.AI_CODE := 16#770A;
   AI_770A.___________0020_0 := false;
   AI_770A.___________0010_2 := false;
   AI_770A.RAW_MIN := -6000;
   AI_770A.RAW_MAX := 13000;
   AI_770A.RAW_NAME := 'Thermal Resistance - 4-wire (Ni1000 climate - 617)';
   AI_770A.___________0030_1 := false;
   AI_770A.___________0030_2 := false;
   AI_770A.PARAM_TYPE := 16#07;
   AI_770A.PARAM_RANGE := 16#0A;
   AI_770A.PARAM_COEF := 16#07;
   AI_770A.VALUE_COEF := 0.00617;
   AI_780A.AI_CODE := 16#780A;
   AI_780A.___________0020_0 := false;
   AI_780A.___________0010_2 := false;
   AI_780A.RAW_MIN := -6000;
   AI_780A.RAW_MAX := 13000;
   AI_780A.RAW_NAME := 'Thermal Resistance - 4-wire (Ni1000 climate - 618)';
   AI_780A.___________0030_1 := false;
   AI_780A.___________0030_2 := false;
   AI_780A.PARAM_TYPE := 16#07;
   AI_780A.PARAM_RANGE := 16#0A;
   AI_780A.PARAM_COEF := 16#08;
   AI_780A.VALUE_COEF := 0.00618;
   AI_790A.AI_CODE := 16#790A;
   AI_790A.___________0020_0 := false;
   AI_790A.___________0010_2 := false;
   AI_790A.RAW_MIN := -6000;
   AI_790A.RAW_MAX := 13000;
   AI_790A.RAW_NAME := 'Thermal Resistance - 4-wire (Ni1000 climate - 672)';
   AI_790A.___________0030_1 := false;
   AI_790A.___________0030_2 := false;
   AI_790A.PARAM_TYPE := 16#07;
   AI_790A.PARAM_RANGE := 16#0A;
   AI_790A.PARAM_COEF := 16#09;
   AI_790A.VALUE_COEF := 0.00672;
   AI_7706.AI_CODE := 16#7706;
   AI_7706.___________0020_0 := false;
   AI_7706.___________0010_2 := false;
   AI_7706.RAW_MIN := -600;
   AI_7706.RAW_MAX := 1800;
   AI_7706.RAW_NAME := 'Thermal Resistance - 4-wire (Ni1000 standard - 617)';
   AI_7706.___________0030_1 := false;
   AI_7706.___________0030_2 := false;
   AI_7706.PARAM_TYPE := 16#07;
   AI_7706.PARAM_RANGE := 16#06;
   AI_7706.PARAM_COEF := 16#07;
   AI_7706.VALUE_COEF := 0.00617;
   AI_7806.AI_CODE := 16#7806;
   AI_7806.___________0020_0 := false;
   AI_7806.___________0010_2 := false;
   AI_7806.RAW_MIN := -600;
   AI_7806.RAW_MAX := 2500;
   AI_7806.RAW_NAME := 'Thermal Resistance - 4-wire (Ni1000 standard - 618)';
   AI_7806.___________0030_1 := false;
   AI_7806.___________0030_2 := false;
   AI_7806.PARAM_TYPE := 16#07;
   AI_7806.PARAM_RANGE := 16#06;
   AI_7806.PARAM_COEF := 16#08;
   AI_7806.VALUE_COEF := 0.00618;
   AI_7906.AI_CODE := 16#7906;
   AI_7906.___________0020_0 := false;
   AI_7906.___________0010_2 := false;
   AI_7906.RAW_MIN := -600;
   AI_7906.RAW_MAX := 2500;
   AI_7906.RAW_NAME := 'Thermal Resistance - 4-wire (Ni1000 standard - 672)';
   AI_7906.___________0030_1 := false;
   AI_7906.___________0030_2 := false;
   AI_7906.PARAM_TYPE := 16#07;
   AI_7906.PARAM_RANGE := 16#06;
   AI_7906.PARAM_COEF := 16#09;
   AI_7906.VALUE_COEF := 0.00672;
   AI_7015.AI_CODE := 16#7015;
   AI_7015.___________0020_0 := false;
   AI_7015.___________0010_2 := false;
   AI_7015.RAW_MIN := -12000;
   AI_7015.RAW_MAX := 13000;
   AI_7015.RAW_NAME := 'Thermal Resistance - 4-wire (Pt10 climate - 3851)';
   AI_7015.___________0030_1 := false;
   AI_7015.___________0030_2 := false;
   AI_7015.PARAM_TYPE := 16#07;
   AI_7015.PARAM_RANGE := 16#15;
   AI_7015.PARAM_COEF := 16#00;
   AI_7015.VALUE_COEF := 0.003851;
   AI_7215.AI_CODE := 16#7215;
   AI_7215.___________0020_0 := false;
   AI_7215.___________0010_2 := false;
   AI_7215.RAW_MIN := -12000;
   AI_7215.RAW_MAX := 13000;
   AI_7215.RAW_NAME := 'Thermal Resistance - 4-wire (Pt10 climate - 3902)';
   AI_7215.___________0030_1 := false;
   AI_7215.___________0030_2 := false;
   AI_7215.PARAM_TYPE := 16#07;
   AI_7215.PARAM_RANGE := 16#15;
   AI_7215.PARAM_COEF := 16#02;
   AI_7215.VALUE_COEF := 0.003902;
   AI_7515.AI_CODE := 16#7515;
   AI_7515.___________0020_0 := false;
   AI_7515.___________0010_2 := false;
   AI_7515.RAW_MIN := -12000;
   AI_7515.RAW_MAX := 13000;
   AI_7515.RAW_NAME := 'Thermal Resistance - 4-wire (Pt10 climate - 391)';
   AI_7515.___________0030_1 := false;
   AI_7515.___________0030_2 := false;
   AI_7515.PARAM_TYPE := 16#07;
   AI_7515.PARAM_RANGE := 16#15;
   AI_7515.PARAM_COEF := 16#05;
   AI_7515.VALUE_COEF := 0.00391;
   AI_7115.AI_CODE := 16#7115;
   AI_7115.___________0020_0 := false;
   AI_7115.___________0010_2 := false;
   AI_7115.RAW_MIN := -12000;
   AI_7115.RAW_MAX := 13000;
   AI_7115.RAW_NAME := 'Thermal Resistance - 4-wire (Pt10 climate - 3916)';
   AI_7115.___________0030_1 := false;
   AI_7115.___________0030_2 := false;
   AI_7115.PARAM_TYPE := 16#07;
   AI_7115.PARAM_RANGE := 16#15;
   AI_7115.PARAM_COEF := 16#01;
   AI_7115.VALUE_COEF := 0.003916;
   AI_7315.AI_CODE := 16#7315;
   AI_7315.___________0020_0 := false;
   AI_7315.___________0010_2 := false;
   AI_7315.RAW_MIN := -12000;
   AI_7315.RAW_MAX := 13000;
   AI_7315.RAW_NAME := 'Thermal Resistance - 4-wire (Pt10 climate - 392)';
   AI_7315.___________0030_1 := false;
   AI_7315.___________0030_2 := false;
   AI_7315.PARAM_TYPE := 16#07;
   AI_7315.PARAM_RANGE := 16#15;
   AI_7315.PARAM_COEF := 16#03;
   AI_7315.VALUE_COEF := 0.00392;
   AI_7014.AI_CODE := 16#7014;
   AI_7014.___________0020_0 := false;
   AI_7014.___________0010_2 := false;
   AI_7014.RAW_MIN := -2000;
   AI_7014.RAW_MAX := 8500;
   AI_7014.RAW_NAME := 'Thermal Resistance - 4-wire (Pt10 standard - 3851)';
   AI_7014.___________0030_1 := false;
   AI_7014.___________0030_2 := false;
   AI_7014.PARAM_TYPE := 16#07;
   AI_7014.PARAM_RANGE := 16#14;
   AI_7014.PARAM_COEF := 16#00;
   AI_7014.VALUE_COEF := 0.003851;
   AI_7214.AI_CODE := 16#7214;
   AI_7214.___________0020_0 := false;
   AI_7214.___________0010_2 := false;
   AI_7214.RAW_MIN := -2000;
   AI_7214.RAW_MAX := 8500;
   AI_7214.RAW_NAME := 'Thermal Resistance - 4-wire (Pt10 standard - 3902)';
   AI_7214.___________0030_1 := false;
   AI_7214.___________0030_2 := false;
   AI_7214.PARAM_TYPE := 16#07;
   AI_7214.PARAM_RANGE := 16#14;
   AI_7214.PARAM_COEF := 16#02;
   AI_7214.VALUE_COEF := 0.003902;
   AI_7514.AI_CODE := 16#7514;
   AI_7514.___________0020_0 := false;
   AI_7514.___________0010_2 := false;
   AI_7514.RAW_MIN := -2000;
   AI_7514.RAW_MAX := 8500;
   AI_7514.RAW_NAME := 'Thermal Resistance - 4-wire (Pt10 standard - 391)';
   AI_7514.___________0030_1 := false;
   AI_7514.___________0030_2 := false;
   AI_7514.PARAM_TYPE := 16#07;
   AI_7514.PARAM_RANGE := 16#14;
   AI_7514.PARAM_COEF := 16#05;
   AI_7514.VALUE_COEF := 0.00391;
   AI_7114.AI_CODE := 16#7114;
   AI_7114.___________0020_0 := false;
   AI_7114.___________0010_2 := false;
   AI_7114.RAW_MIN := -2000;
   AI_7114.RAW_MAX := 8500;
   AI_7114.RAW_NAME := 'Thermal Resistance - 4-wire (Pt10 standard - 3916)';
   AI_7114.___________0030_1 := false;
   AI_7114.___________0030_2 := false;
   AI_7114.PARAM_TYPE := 16#07;
   AI_7114.PARAM_RANGE := 16#14;
   AI_7114.PARAM_COEF := 16#01;
   AI_7114.VALUE_COEF := 0.003916;
   AI_7314.AI_CODE := 16#7314;
   AI_7314.___________0020_0 := false;
   AI_7314.___________0010_2 := false;
   AI_7314.RAW_MIN := -2000;
   AI_7314.RAW_MAX := 8500;
   AI_7314.RAW_NAME := 'Thermal Resistance - 4-wire (Pt10 standard - 392)';
   AI_7314.___________0030_1 := false;
   AI_7314.___________0030_2 := false;
   AI_7314.PARAM_TYPE := 16#07;
   AI_7314.PARAM_RANGE := 16#14;
   AI_7314.PARAM_COEF := 16#03;
   AI_7314.VALUE_COEF := 0.00392;
   AI_7017.AI_CODE := 16#7017;
   AI_7017.___________0020_0 := false;
   AI_7017.___________0010_2 := false;
   AI_7017.RAW_MIN := -12000;
   AI_7017.RAW_MAX := 13000;
   AI_7017.RAW_NAME := 'Thermal Resistance - 4-wire (Pt50 climate - 3851)';
   AI_7017.___________0030_1 := false;
   AI_7017.___________0030_2 := false;
   AI_7017.PARAM_TYPE := 16#07;
   AI_7017.PARAM_RANGE := 16#17;
   AI_7017.PARAM_COEF := 16#00;
   AI_7017.VALUE_COEF := 0.003851;
   AI_7217.AI_CODE := 16#7217;
   AI_7217.___________0020_0 := false;
   AI_7217.___________0010_2 := false;
   AI_7217.RAW_MIN := -12000;
   AI_7217.RAW_MAX := 13000;
   AI_7217.RAW_NAME := 'Thermal Resistance - 4-wire (Pt50 climate - 3902)';
   AI_7217.___________0030_1 := false;
   AI_7217.___________0030_2 := false;
   AI_7217.PARAM_TYPE := 16#07;
   AI_7217.PARAM_RANGE := 16#17;
   AI_7217.PARAM_COEF := 16#02;
   AI_7217.VALUE_COEF := 0.003902;
   AI_7517.AI_CODE := 16#7517;
   AI_7517.___________0020_0 := false;
   AI_7517.___________0010_2 := false;
   AI_7517.RAW_MIN := -12000;
   AI_7517.RAW_MAX := 13000;
   AI_7517.RAW_NAME := 'Thermal Resistance - 4-wire (Pt50 climate - 391)';
   AI_7517.___________0030_1 := false;
   AI_7517.___________0030_2 := false;
   AI_7517.PARAM_TYPE := 16#07;
   AI_7517.PARAM_RANGE := 16#17;
   AI_7517.PARAM_COEF := 16#05;
   AI_7517.VALUE_COEF := 0.00391;
   AI_7117.AI_CODE := 16#7117;
   AI_7117.___________0020_0 := false;
   AI_7117.___________0010_2 := false;
   AI_7117.RAW_MIN := -12000;
   AI_7117.RAW_MAX := 13000;
   AI_7117.RAW_NAME := 'Thermal Resistance - 4-wire (Pt50 climate - 3916)';
   AI_7117.___________0030_1 := false;
   AI_7117.___________0030_2 := false;
   AI_7117.PARAM_TYPE := 16#07;
   AI_7117.PARAM_RANGE := 16#17;
   AI_7117.PARAM_COEF := 16#01;
   AI_7117.VALUE_COEF := 0.003916;
   AI_7317.AI_CODE := 16#7317;
   AI_7317.___________0020_0 := false;
   AI_7317.___________0010_2 := false;
   AI_7317.RAW_MIN := -12000;
   AI_7317.RAW_MAX := 13000;
   AI_7317.RAW_NAME := 'Thermal Resistance - 4-wire (Pt50 climate - 392)';
   AI_7317.___________0030_1 := false;
   AI_7317.___________0030_2 := false;
   AI_7317.PARAM_TYPE := 16#07;
   AI_7317.PARAM_RANGE := 16#17;
   AI_7317.PARAM_COEF := 16#03;
   AI_7317.VALUE_COEF := 0.00392;
   AI_7016.AI_CODE := 16#7016;
   AI_7016.___________0020_0 := false;
   AI_7016.___________0010_2 := false;
   AI_7016.RAW_MIN := -2000;
   AI_7016.RAW_MAX := 8500;
   AI_7016.RAW_NAME := 'Thermal Resistance - 4-wire (Pt50 standard - 3851)';
   AI_7016.___________0030_1 := false;
   AI_7016.___________0030_2 := false;
   AI_7016.PARAM_TYPE := 16#07;
   AI_7016.PARAM_RANGE := 16#16;
   AI_7016.PARAM_COEF := 16#00;
   AI_7016.VALUE_COEF := 0.003851;
   AI_7216.AI_CODE := 16#7216;
   AI_7216.___________0020_0 := false;
   AI_7216.___________0010_2 := false;
   AI_7216.RAW_MIN := -2000;
   AI_7216.RAW_MAX := 8500;
   AI_7216.RAW_NAME := 'Thermal Resistance - 4-wire (Pt50 standard - 3902)';
   AI_7216.___________0030_1 := false;
   AI_7216.___________0030_2 := false;
   AI_7216.PARAM_TYPE := 16#07;
   AI_7216.PARAM_RANGE := 16#16;
   AI_7216.PARAM_COEF := 16#02;
   AI_7216.VALUE_COEF := 0.003902;
   AI_7516.AI_CODE := 16#7516;
   AI_7516.___________0020_0 := false;
   AI_7516.___________0010_2 := false;
   AI_7516.RAW_MIN := -2000;
   AI_7516.RAW_MAX := 8500;
   AI_7516.RAW_NAME := 'Thermal Resistance - 4-wire (Pt50 standard - 391)';
   AI_7516.___________0030_1 := false;
   AI_7516.___________0030_2 := false;
   AI_7516.PARAM_TYPE := 16#07;
   AI_7516.PARAM_RANGE := 16#16;
   AI_7516.PARAM_COEF := 16#05;
   AI_7516.VALUE_COEF := 0.00391;
   AI_7116.AI_CODE := 16#7116;
   AI_7116.___________0020_0 := false;
   AI_7116.___________0010_2 := false;
   AI_7116.RAW_MIN := -2000;
   AI_7116.RAW_MAX := 8500;
   AI_7116.RAW_NAME := 'Thermal Resistance - 4-wire (Pt50 standard - 3916)';
   AI_7116.___________0030_1 := false;
   AI_7116.___________0030_2 := false;
   AI_7116.PARAM_TYPE := 16#07;
   AI_7116.PARAM_RANGE := 16#16;
   AI_7116.PARAM_COEF := 16#01;
   AI_7116.VALUE_COEF := 0.003916;
   AI_7316.AI_CODE := 16#7316;
   AI_7316.___________0020_0 := false;
   AI_7316.___________0010_2 := false;
   AI_7316.RAW_MIN := -2000;
   AI_7316.RAW_MAX := 8500;
   AI_7316.RAW_NAME := 'Thermal Resistance - 4-wire (Pt50 standard - 392)';
   AI_7316.___________0030_1 := false;
   AI_7316.___________0030_2 := false;
   AI_7316.PARAM_TYPE := 16#07;
   AI_7316.PARAM_RANGE := 16#16;
   AI_7316.PARAM_COEF := 16#03;
   AI_7316.VALUE_COEF := 0.00392;
   AI_7000.AI_CODE := 16#7000;
   AI_7000.___________0020_0 := false;
   AI_7000.___________0010_2 := false;
   AI_7000.RAW_MIN := -12000;
   AI_7000.RAW_MAX := 13000;
   AI_7000.RAW_NAME := 'Thermal Resistance - 4-wire (Pt100 climate - 3851)';
   AI_7000.___________0030_1 := false;
   AI_7000.___________0030_2 := false;
   AI_7000.PARAM_TYPE := 16#07;
   AI_7000.PARAM_RANGE := 16#00;
   AI_7000.PARAM_COEF := 16#00;
   AI_7000.VALUE_COEF := 0.003851;
   AI_7200.AI_CODE := 16#7200;
   AI_7200.___________0020_0 := false;
   AI_7200.___________0010_2 := false;
   AI_7200.RAW_MIN := -12000;
   AI_7200.RAW_MAX := 13000;
   AI_7200.RAW_NAME := 'Thermal Resistance - 4-wire (Pt100 climate - 3902)';
   AI_7200.___________0030_1 := false;
   AI_7200.___________0030_2 := false;
   AI_7200.PARAM_TYPE := 16#07;
   AI_7200.PARAM_RANGE := 16#00;
   AI_7200.PARAM_COEF := 16#02;
   AI_7200.VALUE_COEF := 0.003902;
   AI_7500.AI_CODE := 16#7500;
   AI_7500.___________0020_0 := false;
   AI_7500.___________0010_2 := false;
   AI_7500.RAW_MIN := -12000;
   AI_7500.RAW_MAX := 13000;
   AI_7500.RAW_NAME := 'Thermal Resistance - 4-wire (Pt100 climate - 391)';
   AI_7500.___________0030_1 := false;
   AI_7500.___________0030_2 := false;
   AI_7500.PARAM_TYPE := 16#07;
   AI_7500.PARAM_RANGE := 16#00;
   AI_7500.PARAM_COEF := 16#05;
   AI_7500.VALUE_COEF := 0.00391;
   AI_7100.AI_CODE := 16#7100;
   AI_7100.___________0020_0 := false;
   AI_7100.___________0010_2 := false;
   AI_7100.RAW_MIN := -12000;
   AI_7100.RAW_MAX := 13000;
   AI_7100.RAW_NAME := 'Thermal Resistance - 4-wire (Pt100 climate - 3916)';
   AI_7100.___________0030_1 := false;
   AI_7100.___________0030_2 := false;
   AI_7100.PARAM_TYPE := 16#07;
   AI_7100.PARAM_RANGE := 16#00;
   AI_7100.PARAM_COEF := 16#01;
   AI_7100.VALUE_COEF := 0.003916;
   AI_7300.AI_CODE := 16#7300;
   AI_7300.___________0020_0 := false;
   AI_7300.___________0010_2 := false;
   AI_7300.RAW_MIN := -12000;
   AI_7300.RAW_MAX := 13000;
   AI_7300.RAW_NAME := 'Thermal Resistance - 4-wire (Pt100 climate - 392)';
   AI_7300.___________0030_1 := false;
   AI_7300.___________0030_2 := false;
   AI_7300.PARAM_TYPE := 16#07;
   AI_7300.PARAM_RANGE := 16#00;
   AI_7300.PARAM_COEF := 16#03;
   AI_7300.VALUE_COEF := 0.00392;
   AI_7002.AI_CODE := 16#7002;
   AI_7002.___________0020_0 := false;
   AI_7002.___________0010_2 := false;
   AI_7002.RAW_MIN := -2000;
   AI_7002.RAW_MAX := 8500;
   AI_7002.RAW_NAME := 'Thermal Resistance - 4-wire (Pt100 standard - 3851)';
   AI_7002.___________0030_1 := false;
   AI_7002.___________0030_2 := false;
   AI_7002.PARAM_TYPE := 16#07;
   AI_7002.PARAM_RANGE := 16#02;
   AI_7002.PARAM_COEF := 16#00;
   AI_7002.VALUE_COEF := 0.003851;
   AI_7202.AI_CODE := 16#7202;
   AI_7202.___________0020_0 := false;
   AI_7202.___________0010_2 := false;
   AI_7202.RAW_MIN := -2000;
   AI_7202.RAW_MAX := 8500;
   AI_7202.RAW_NAME := 'Thermal Resistance - 4-wire (Pt100 standard - 3902)';
   AI_7202.___________0030_1 := false;
   AI_7202.___________0030_2 := false;
   AI_7202.PARAM_TYPE := 16#07;
   AI_7202.PARAM_RANGE := 16#02;
   AI_7202.PARAM_COEF := 16#02;
   AI_7202.VALUE_COEF := 0.003902;
   AI_7502.AI_CODE := 16#7502;
   AI_7502.___________0020_0 := false;
   AI_7502.___________0010_2 := false;
   AI_7502.RAW_MIN := -2000;
   AI_7502.RAW_MAX := 8500;
   AI_7502.RAW_NAME := 'Thermal Resistance - 4-wire (Pt100 standard - 391)';
   AI_7502.___________0030_1 := false;
   AI_7502.___________0030_2 := false;
   AI_7502.PARAM_TYPE := 16#07;
   AI_7502.PARAM_RANGE := 16#02;
   AI_7502.PARAM_COEF := 16#05;
   AI_7502.VALUE_COEF := 0.00391;
   AI_7102.AI_CODE := 16#7102;
   AI_7102.___________0020_0 := false;
   AI_7102.___________0010_2 := false;
   AI_7102.RAW_MIN := -2000;
   AI_7102.RAW_MAX := 8500;
   AI_7102.RAW_NAME := 'Thermal Resistance - 4-wire (Pt100 standard - 3916)';
   AI_7102.___________0030_1 := false;
   AI_7102.___________0030_2 := false;
   AI_7102.PARAM_TYPE := 16#07;
   AI_7102.PARAM_RANGE := 16#02;
   AI_7102.PARAM_COEF := 16#01;
   AI_7102.VALUE_COEF := 0.003916;
   AI_7302.AI_CODE := 16#7302;
   AI_7302.___________0020_0 := false;
   AI_7302.___________0010_2 := false;
   AI_7302.RAW_MIN := -2000;
   AI_7302.RAW_MAX := 8500;
   AI_7302.RAW_NAME := 'Thermal Resistance - 4-wire (Pt100 standard - 392)';
   AI_7302.___________0030_1 := false;
   AI_7302.___________0030_2 := false;
   AI_7302.PARAM_TYPE := 16#07;
   AI_7302.PARAM_RANGE := 16#02;
   AI_7302.PARAM_COEF := 16#03;
   AI_7302.VALUE_COEF := 0.00392;
   AI_7007.AI_CODE := 16#7007;
   AI_7007.___________0020_0 := false;
   AI_7007.___________0010_2 := false;
   AI_7007.RAW_MIN := -12000;
   AI_7007.RAW_MAX := 13000;
   AI_7007.RAW_NAME := 'Thermal Resistance - 4-wire (Pt200 climate - 3851)';
   AI_7007.___________0030_1 := false;
   AI_7007.___________0030_2 := false;
   AI_7007.PARAM_TYPE := 16#07;
   AI_7007.PARAM_RANGE := 16#07;
   AI_7007.PARAM_COEF := 16#00;
   AI_7007.VALUE_COEF := 0.003851;
   AI_7207.AI_CODE := 16#7207;
   AI_7207.___________0020_0 := false;
   AI_7207.___________0010_2 := false;
   AI_7207.RAW_MIN := -12000;
   AI_7207.RAW_MAX := 13000;
   AI_7207.RAW_NAME := 'Thermal Resistance - 4-wire (Pt200 climate - 3902)';
   AI_7207.___________0030_1 := false;
   AI_7207.___________0030_2 := false;
   AI_7207.PARAM_TYPE := 16#07;
   AI_7207.PARAM_RANGE := 16#07;
   AI_7207.PARAM_COEF := 16#02;
   AI_7207.VALUE_COEF := 0.003902;
   AI_7507.AI_CODE := 16#7507;
   AI_7507.___________0020_0 := false;
   AI_7507.___________0010_2 := false;
   AI_7507.RAW_MIN := -12000;
   AI_7507.RAW_MAX := 13000;
   AI_7507.RAW_NAME := 'Thermal Resistance - 4-wire (Pt200 climate - 391)';
   AI_7507.___________0030_1 := false;
   AI_7507.___________0030_2 := false;
   AI_7507.PARAM_TYPE := 16#07;
   AI_7507.PARAM_RANGE := 16#07;
   AI_7507.PARAM_COEF := 16#05;
   AI_7507.VALUE_COEF := 0.00391;
   AI_7107.AI_CODE := 16#7107;
   AI_7107.___________0020_0 := false;
   AI_7107.___________0010_2 := false;
   AI_7107.RAW_MIN := -12000;
   AI_7107.RAW_MAX := 13000;
   AI_7107.RAW_NAME := 'Thermal Resistance - 4-wire (Pt200 climate - 3916)';
   AI_7107.___________0030_1 := false;
   AI_7107.___________0030_2 := false;
   AI_7107.PARAM_TYPE := 16#07;
   AI_7107.PARAM_RANGE := 16#07;
   AI_7107.PARAM_COEF := 16#01;
   AI_7107.VALUE_COEF := 0.003916;
   AI_7307.AI_CODE := 16#7307;
   AI_7307.___________0020_0 := false;
   AI_7307.___________0010_2 := false;
   AI_7307.RAW_MIN := -12000;
   AI_7307.RAW_MAX := 13000;
   AI_7307.RAW_NAME := 'Thermal Resistance - 4-wire (Pt200 climate - 392)';
   AI_7307.___________0030_1 := false;
   AI_7307.___________0030_2 := false;
   AI_7307.PARAM_TYPE := 16#07;
   AI_7307.PARAM_RANGE := 16#07;
   AI_7307.PARAM_COEF := 16#03;
   AI_7307.VALUE_COEF := 0.00392;
   AI_700B.AI_CODE := 16#700B;
   AI_700B.___________0020_0 := false;
   AI_700B.___________0010_2 := false;
   AI_700B.RAW_MIN := -2000;
   AI_700B.RAW_MAX := 8500;
   AI_700B.RAW_NAME := 'Thermal Resistance - 4-wire (Pt200 standard - 3851)';
   AI_700B.___________0030_1 := false;
   AI_700B.___________0030_2 := false;
   AI_700B.PARAM_TYPE := 16#07;
   AI_700B.PARAM_RANGE := 16#0B;
   AI_700B.PARAM_COEF := 16#00;
   AI_700B.VALUE_COEF := 0.003851;
   AI_720B.AI_CODE := 16#720B;
   AI_720B.___________0020_0 := false;
   AI_720B.___________0010_2 := false;
   AI_720B.RAW_MIN := -2000;
   AI_720B.RAW_MAX := 8500;
   AI_720B.RAW_NAME := 'Thermal Resistance - 4-wire (Pt200 standard - 3902)';
   AI_720B.___________0030_1 := false;
   AI_720B.___________0030_2 := false;
   AI_720B.PARAM_TYPE := 16#07;
   AI_720B.PARAM_RANGE := 16#0B;
   AI_720B.PARAM_COEF := 16#02;
   AI_720B.VALUE_COEF := 0.003902;
   AI_750B.AI_CODE := 16#750B;
   AI_750B.___________0020_0 := false;
   AI_750B.___________0010_2 := false;
   AI_750B.RAW_MIN := -2000;
   AI_750B.RAW_MAX := 8500;
   AI_750B.RAW_NAME := 'Thermal Resistance - 4-wire (Pt200 standard - 391)';
   AI_750B.___________0030_1 := false;
   AI_750B.___________0030_2 := false;
   AI_750B.PARAM_TYPE := 16#07;
   AI_750B.PARAM_RANGE := 16#0B;
   AI_750B.PARAM_COEF := 16#05;
   AI_750B.VALUE_COEF := 0.00391;
   AI_710B.AI_CODE := 16#710B;
   AI_710B.___________0020_0 := false;
   AI_710B.___________0010_2 := false;
   AI_710B.RAW_MIN := -2000;
   AI_710B.RAW_MAX := 8500;
   AI_710B.RAW_NAME := 'Thermal Resistance - 4-wire (Pt200 standard - 3916)';
   AI_710B.___________0030_1 := false;
   AI_710B.___________0030_2 := false;
   AI_710B.PARAM_TYPE := 16#07;
   AI_710B.PARAM_RANGE := 16#0B;
   AI_710B.PARAM_COEF := 16#01;
   AI_710B.VALUE_COEF := 0.003916;
   AI_730B.AI_CODE := 16#730B;
   AI_730B.___________0020_0 := false;
